# B&R Automation Studio project OpcUaSample410_BrbLibUa103 (part 20)

#### Main.st - Init, cyclic, exit code
```iecst
PROGRAM _INIT
	brsmemset(ADR(Opc), 0, SIZEOF(Opc));
	Opc.OwnGetCertificateList.fbUaSrv_MethodOperate.MethodName := 'OwnGetCertificateList'; // Name der Methode wie in 'Methods.uam' angegeben
	Opc.OwnGenerate.fbUaSrv_MethodOperate.MethodName := 'OwnGenerate'; // Name der Methode wie in 'Methods.uam' angegeben
	Opc.OwnImport.fbUaSrv_MethodOperate.MethodName := 'OwnImport'; // Name der Methode wie in 'Methods.uam' angegeben
	Opc.OwnDelete.fbUaSrv_MethodOperate.MethodName := 'OwnDelete'; // Name der Methode wie in 'Methods.uam' angegeben

	Opc.ForeignGetCertificateList.fbUaSrv_MethodOperate.MethodName := 'ForeignGetCertificateList'; // Name der Methode wie in 'Methods.uam' angegeben
	Opc.ForeignImport.fbUaSrv_MethodOperate.MethodName := 'ForeignImport'; // Name der Methode wie in 'Methods.uam' angegeben
	Opc.ForeignDelete.fbUaSrv_MethodOperate.MethodName := 'ForeignDelete'; // Name der Methode wie in 'Methods.uam' angegeben

	Opc.SslGetCfgList.fbUaSrv_MethodOperate.MethodName := 'SslGetCfgList'; // Name der Methode wie in 'Methods.uam' angegeben
	Opc.SslGetTrustedCertList.fbUaSrv_MethodOperate.MethodName := 'SslGetTrustedCertList'; // Name der Methode wie in 'Methods.uam' angegeben

	Opc.Warmstart.fbUaSrv_MethodOperate.MethodName := 'Warmstart'; // Name der Methode wie in 'Methods.uam' angegeben
END_PROGRAM

PROGRAM _CYCLIC
	// Methode 'OwnGetCertificateList'
	CASE Opc.OwnGetCertificateList.Step.nStepNr OF
		0:	// Prüfen, ob Methode von einem Client aufgerufen wurde
			Opc.OwnGetCertificateList.fbUaSrv_MethodOperate.Execute := 1;
			Opc.OwnGetCertificateList.fbUaSrv_MethodOperate.Action := UaMoa_CheckIsCalled;
			IF Opc.OwnGetCertificateList.fbUaSrv_MethodOperate.Done = 1 THEN
				Opc.OwnGetCertificateList.fbUaSrv_MethodOperate.Execute := 0;
				IF Opc.OwnGetCertificateList.fbUaSrv_MethodOperate.IsCalled = 1 THEN
					// Variablen der Eingans-Argumente sind besetzt -> Methode ausführen
					Opc.OwnGetCertificateList.nCallCount := Opc.OwnGetCertificateList.nCallCount + 1;	// Nur zur Diagnose
					Opc.OwnGetCertificateList.Out_ErrorId := 0;
					Opc.OwnGetCertificateList.Step.nStepNr := Opc.OwnGetCertificateList.Step.nStepNr + 1;
				END_IF
			ELSIF Opc.OwnGetCertificateList.fbUaSrv_MethodOperate.Error = 1 THEN
					Opc.OwnGetCertificateList.fbUaSrv_MethodOperate.Execute := 0;
				Opc.OwnGetCertificateList.Step.nErrorStep := Opc.OwnGetCertificateList.Step.nStepNr;
				Opc.OwnGetCertificateList.Step.eAction := Opc.OwnGetCertificateList.fbUaSrv_MethodOperate.Action;
				Opc.OwnGetCertificateList.Step.nErrorId := Opc.OwnGetCertificateList.fbUaSrv_MethodOperate.ErrorID;
			END_IF

		1:	// Vorbereitung zum Auslesen der Liste
			Opc.OwnGetCertificateList.fbArCertGetOwnDetails.Execute := 0;
			Opc.OwnGetCertificateList.fbArCertGetOwnDetails.Name := '';
			Opc.OwnGetCertificateList.fbArCertGetOwnDetails.Index := 0;
			brsmemset(ADR(Opc.OwnGetCertificateList.Out_CertificatesList), 0, SIZEOF(Opc.OwnGetCertificateList.Out_CertificatesList));
			Opc.OwnGetCertificateList.Step.nStepNr := Opc.OwnGetCertificateList.Step.nStepNr + 1;

		2:	// Nächsten Eintrag auslesen
			IF Opc.OwnGetCertificateList.Out_CertificatesList.nLength <= OPCUA_CERTS_INDEX_MAX THEN
				Opc.OwnGetCertificateList.fbArCertGetOwnDetails.Execute := 1;
				IF Opc.OwnGetCertificateList.fbArCertGetOwnDetails.Busy = 0 THEN
					IF Opc.OwnGetCertificateList.fbArCertGetOwnDetails.Done = 1 THEN
						// Eintrag auf Ausgangs-Argument übertragen
						brsmemcpy(ADR(Opc.OwnGetCertificateList.Out_CertificatesList.Data[Opc.OwnGetCertificateList.Out_CertificatesList.nLength]), ADR(Opc.OwnGetCertificateList.fbArCertGetOwnDetails.Details), SIZEOF(ArCertDetailsType));
						// Nächsten Eintrag lesen
						Opc.OwnGetCertificateList.Out_CertificatesList.nLength := Opc.OwnGetCertificateList.Out_CertificatesList.nLength + 1;
						Opc.OwnGetCertificateList.fbArCertGetOwnDetails.Index := Opc.OwnGetCertificateList.Out_CertificatesList.nLength;
						Opc.OwnGetCertificateList.fbArCertGetOwnDetails.Execute := 0;
					ELSIF Opc.OwnGetCertificateList.fbArCertGetOwnDetails.Error = 1 THEN
						IF Opc.OwnGetCertificateList.fbArCertGetOwnDetails.StatusID = arCERT_ERR_CERTIFICATE_NOT_FOUND THEN
							// Alle Einträge sind gelesen
							Opc.OwnGetCertificateList.fbArCertGetOwnDetails.Execute := 0;
							Opc.OwnGetCertificateList.Step.nStepNr := Opc.OwnGetCertificateList.Step.nStepNr + 1;
						ELSE
							// Fehler beim Auslesen
							Opc.OwnGetCertificateList.fbArCertGetOwnDetails.Execute := 0;
							Opc.OwnGetCertificateList.Out_ErrorId := Opc.OwnGetCertificateList.fbArCertGetOwnDetails.StatusID;
							Opc.OwnGetCertificateList.Step.nStepNr := Opc.OwnGetCertificateList.Step.nStepNr + 1;
						END_IF
					END_IF
				END_IF
			ELSE
				// Das SPS-Array ist nicht genügend groß, um weitere Einträge aufzunehmen
				Opc.OwnGetCertificateList.Out_ErrorId := 12189696; // := 0x00BA0000 := Good_ResultsMayBeIncomplete
				Opc.OwnGetCertificateList.Step.nStepNr := Opc.OwnGetCertificateList.Step.nStepNr + 1;
			END_IF

		3:	// Rückmelden, dass Methode ausgeführt wurde
			Opc.OwnGetCertificateList.fbUaSrv_MethodOperate.Execute := 1;
			Opc.OwnGetCertificateList.fbUaSrv_MethodOperate.Action := UaMoa_Finished;
			IF Opc.OwnGetCertificateList.fbUaSrv_MethodOperate.Done = 1 THEN
				Opc.OwnGetCertificateList.fbUaSrv_MethodOperate.Execute := 0;
				Opc.OwnGetCertificateList.Step.nStepNr := 0;
			ELSIF Opc.OwnGetCertificateList.fbUaSrv_MethodOperate.Error = 1 THEN
				// Fehler eintragen, aber trotzdem weiter machen
				Opc.OwnGetCertificateList.fbUaSrv_MethodOperate.Execute := 0;
				Opc.OwnGetCertificateList.Step.nErrorStep := Opc.OwnGetCertificateList.Step.nStepNr;
				Opc.OwnGetCertificateList.Step.eAction := Opc.OwnGetCertificateList.fbUaSrv_MethodOperate.Action;
				Opc.OwnGetCertificateList.Step.nErrorId := Opc.OwnGetCertificateList.fbUaSrv_MethodOperate.ErrorID;
				Opc.OwnGetCertificateList.Step.nStepNr := 0;
			END_IF

	END_CASE
	Opc.OwnGetCertificateList.fbUaSrv_MethodOperate();
	Opc.OwnGetCertificateList.fbArCertGetOwnDetails();

		// Methode 'OwnGenerate'
	CASE Opc.OwnGenerate.Step.nStepNr OF
		0:	// Prüfen, ob Methode von einem Client aufgerufen wurde
			Opc.OwnGenerate.fbUaSrv_MethodOperate.Execute := 1;
			Opc.OwnGenerate.fbUaSrv_MethodOperate.Action := UaMoa_CheckIsCalled;
			IF Opc.OwnGenerate.fbUaSrv_MethodOperate.Done = 1 THEN
				Opc.OwnGenerate.fbUaSrv_MethodOperate.Execute := 0;
				IF Opc.OwnGenerate.fbUaSrv_MethodOperate.IsCalled = 1 THEN
					// Variablen der Eingans-Argumente sind besetzt -> Methode ausführen
					Opc.OwnGenerate.nCallCount := Opc.OwnGenerate.nCallCount + 1;	// Nur zur Diagnose
					Opc.OwnGenerate.Out_ErrorId := 0;
					Opc.OwnGenerate.Step.nStepNr := Opc.OwnGenerate.Step.nStepNr + 1;
				END_IF
			ELSIF Opc.OwnGenerate.fbUaSrv_MethodOperate.Error = 1 THEN
				Opc.OwnGenerate.fbUaSrv_MethodOperate.Execute := 0;
				Opc.OwnGenerate.Step.nErrorStep := Opc.OwnGenerate.Step.nStepNr;
				Opc.OwnGenerate.Step.eAction := Opc.OwnGenerate.fbUaSrv_MethodOperate.Action;
				Opc.OwnGenerate.Step.nErrorId := Opc.OwnGenerate.fbUaSrv_MethodOperate.ErrorID;
			END_IF

		1:	// Vorbereitung zum Erzeugen des OpcUa-Zertifikats
			Opc.OwnGenerate.fbArCertGenerateX.Execute := 0;
			Opc.OwnGenerate.fbArCertGenerateX.Name := Opc.OwnGenerate.In_Parameter.sName;
			Opc.OwnGenerate.fbArCertGenerateX.PrivateKeyName := Opc.OwnGenerate.In_Parameter.sPrivateKeyName;
			Opc.OwnGenerate.fbArCertGenerateX.PrivateKeyPassword := Opc.OwnGenerate.In_Parameter.sPrivateKeyPassword;
			Opc.OwnGenerate.fbArCertGenerateX.KeySize := Opc.OwnGenerate.In_Parameter.eKeySize;
			Opc.OwnGenerate.fbArCertGenerateX.CountryCode := Opc.OwnGenerate.In_Parameter.sCountryCode;
			Opc.OwnGenerate.fbArCertGenerateX.StateProvince := Opc.OwnGenerate.In_Parameter.sStateProvince;
			Opc.OwnGenerate.fbArCertGenerateX.Locality := Opc.OwnGenerate.In_Parameter.sLocality;
			Opc.OwnGenerate.fbArCertGenerateX.Organization := Opc.OwnGenerate.In_Parameter.sOrganization;
			Opc.OwnGenerate.fbArCertGenerateX.OrganizationUnit := Opc.OwnGenerate.In_Parameter.sOrganizationUnit;
			Opc.OwnGenerate.fbArCertGenerateX.ContactEmail := Opc.OwnGenerate.In_Parameter.sContactEmail;
			Opc.OwnGenerate.fbArCertGenerateX.CommonName := Opc.OwnGenerate.In_Parameter.sCommonName;
			Opc.OwnGenerate.fbArCertGenerateX.ValidTimeSeconds := Opc.OwnGenerate.In_Parameter.nValidTimeSeconds;
			Opc.OwnGenerate.fbArCertGenerateX.URI := Opc.OwnGenerate.In_Parameter.sUri;
			Opc.OwnGenerate.fbArCertGenerateX.DnsName := Opc.OwnGenerate.In_Parameter.sDnsName;
			Opc.OwnGenerate.fbArCertGenerateX.IP := Opc.OwnGenerate.In_Parameter.sIp;
			Opc.OwnGenerate.Step.nStepNr := Opc.OwnGenerate.Step.nStepNr + 1;

		2:	// Erzeugen des OpcUa-Zertifikats
			Opc.OwnGenerate.fbArCertGenerateX.Execute := 1;
			IF Opc.OwnGenerate.fbArCertGenerateX.Busy = 0 THEN
				IF Opc.OwnGenerate.fbArCertGenerateX.Done = 1 THEN
					// Zertifikat wurde erstellt
					Opc.OwnGenerate.fbArCertGenerateX.Execute := 0;
					Opc.OwnGenerate.Step.nStepNr := Opc.OwnGenerate.Step.nStepNr + 1;
				ELSIF Opc.OwnGenerate.fbArCertGenerateX.Error = 1 THEN
					// Fehler beim Erstellen
					Opc.OwnGenerate.fbArCertGenerateX.Execute := 0;
					Opc.OwnGenerate.Out_ErrorId := Opc.OwnGenerate.fbArCertGenerateX.StatusID;
					Opc.OwnGenerate.Step.nStepNr := Opc.OwnGenerate.Step.nStepNr + 1;
				END_IF
			END_IF

		3:	// Rückmelden, dass Methode ausgeführt wurde
			Opc.OwnGenerate.fbUaSrv_MethodOperate.Execute := 1;
			Opc.OwnGenerate.fbUaSrv_MethodOperate.Action := UaMoa_Finished;
			IF Opc.OwnGenerate.fbUaSrv_MethodOperate.Done = 1 THEN
				Opc.OwnGenerate.fbUaSrv_MethodOperate.Execute := 0;
				Opc.OwnGenerate.Step.nStepNr := 0;
			ELSIF Opc.OwnGenerate.fbUaSrv_MethodOperate.Error = 1 THEN
				// Fehler eintragen, aber trotzdem weiter machen
				Opc.OwnGenerate.fbUaSrv_MethodOperate.Execute := 0;
				Opc.OwnGenerate.Step.nErrorStep := Opc.OwnGenerate.Step.nStepNr;
				Opc.OwnGenerate.Step.eAction := Opc.OwnGenerate.fbUaSrv_MethodOperate.Action;
				Opc.OwnGenerate.Step.nErrorId := Opc.OwnGenerate.fbUaSrv_MethodOperate.ErrorID;
				Opc.OwnGenerate.Step.nStepNr := 0;
			END_IF

	END_CASE
	Opc.OwnGenerate.fbUaSrv_MethodOperate();
	Opc.OwnGenerate.fbArCertGenerateX();

	// Methode 'OwnImport'
	CASE Opc.OwnImport.Step.nStepNr OF
		0:	// Prüfen, ob Methode von einem Client aufgerufen wurde
			Opc.OwnImport.fbUaSrv_MethodOperate.Execute := 1;
			Opc.OwnImport.fbUaSrv_MethodOperate.Action := UaMoa_CheckIsCalled;
			IF Opc.OwnImport.fbUaSrv_MethodOperate.Done = 1 THEN
				Opc.OwnImport.fbUaSrv_MethodOperate.Execute := 0;
				IF Opc.OwnImport.fbUaSrv_MethodOperate.IsCalled = 1 THEN
					// Variablen der Eingans-Argumente sind besetzt -> Methode ausführen
					Opc.OwnImport.nCallCount := Opc.OwnImport.nCallCount + 1;	// Nur zur Diagnose
					Opc.OwnImport.Out_ErrorId := 0;
					Opc.OwnImport.Step.nStepNr := Opc.OwnImport.Step.nStepNr + 1;
				END_IF
			ELSIF Opc.OwnImport.fbUaSrv_MethodOperate.Error = 1 THEN
				Opc.OwnImport.fbUaSrv_MethodOperate.Execute := 0;
				Opc.OwnImport.Step.nErrorStep := Opc.OwnImport.Step.nStepNr;
				Opc.OwnImport.Step.eAction := Opc.OwnImport.fbUaSrv_MethodOperate.Action;
				Opc.OwnImport.Step.nErrorId := Opc.OwnImport.fbUaSrv_MethodOperate.ErrorID;
			END_IF

		1:	// Vorbereitung zum Löschen des öffentlichen Zertifikats
			Opc.OwnImport.fbArCertDeleteOwn.Execute := 0;
			IF Opc.OwnImport.In_Overwrite = 1 THEN
				Opc.OwnImport.fbArCertDeleteOwn.Name := Opc.OwnImport.In_Name;
				Opc.OwnImport.Step.nStepNr := Opc.OwnImport.Step.nStepNr + 1;
			ELSE
				Opc.OwnImport.Step.nStepNr := Opc.OwnImport.Step.nStepNr + 2;
			END_IF

		2:	// Löschen des öffentlichen Zertifikats
			Opc.OwnImport.fbArCertDeleteOwn.Execute := 1;
			IF Opc.OwnImport.fbArCertDeleteOwn.Busy = 0 THEN
				IF Opc.OwnImport.fbArCertDeleteOwn.Done = 1 THEN
					// Zertifikat wurde gelöscht
					Opc.OwnImport.fbArCertDeleteOwn.Execute := 0;
					Opc.OwnImport.Step.nStepNr := Opc.OwnImport.Step.nStepNr + 1;
				ELSIF Opc.OwnImport.fbArCertDeleteOwn.Error = 1 THEN
					// Zertifikat ist nicht vorhanden. Fehler wird übergangen
					Opc.OwnImport.fbArCertDeleteOwn.Execute := 0;
					Opc.OwnImport.Step.nStepNr := Opc.OwnImport.Step.nStepNr + 1;
				END_IF
			END_IF

		3:	// Vorbereitung zum Importieren des öffentlichen Zertifikats
			Opc.OwnImport.fbArCertImportOwn.Execute := 0;
			Opc.OwnImport.fbArCertImportOwn.Name := Opc.OwnImport.In_Name;
			Opc.OwnImport.fbArCertImportOwn.Data := ADR(Opc.OwnImport.In_Certificate.Data);
			Opc.OwnImport.fbArCertImportOwn.DataSize := Opc.OwnImport.In_Certificate.Length;
			Opc.OwnImport.Step.nStepNr := Opc.OwnImport.Step.nStepNr + 1;

		4:	// Importieren des öffentlichen Zertifikats
			Opc.OwnImport.fbArCertImportOwn.Execute := 1;
			IF Opc.OwnImport.fbArCertImportOwn.Busy = 0 THEN
				IF Opc.OwnImport.fbArCertImportOwn.Done = 1 THEN
					// Zertifikat wurde importiert
					Opc.OwnImport.fbArCertImportOwn.Execute := 0;
					Opc.OwnImport.Step.nStepNr := Opc.OwnImport.Step.nStepNr + 1;
				ELSIF Opc.OwnImport.fbArCertImportOwn.Error = 1 THEN
					// Fehler beim Importieren
					Opc.OwnImport.fbArCertImportOwn.Execute := 0;
					Opc.OwnImport.Out_ErrorId := Opc.OwnImport.fbArCertImportOwn.StatusID;
					Opc.OwnImport.Step.nStepNr := Opc.OwnImport.Step.nStepNr + 1;
				END_IF
			END_IF

		5:	// Vorbereitung zum Löschen des privaten Keys
			Opc.OwnImport.fbArCertDeletePrivateKey.Execute := 0;
			IF Opc.OwnImport.In_Overwrite = 1 THEN
				Opc.OwnImport.fbArCertDeletePrivateKey.Name := Opc.OwnImport.In_PrivateKeyName;
				Opc.OwnImport.Step.nStepNr := Opc.OwnImport.Step.nStepNr + 1;
			ELSE
				Opc.OwnImport.Step.nStepNr := Opc.OwnImport.Step.nStepNr + 2;
			END_IF

		6:	// Löschen des privaten Keys
			Opc.OwnImport.fbArCertDeletePrivateKey.Execute := 1;
			IF Opc.OwnImport.fbArCertDeletePrivateKey.Busy = 0 THEN
				IF Opc.OwnImport.fbArCertDeletePrivateKey.Done = 1 THEN
					// Key wurde gelöscht
					Opc.OwnImport.fbArCertDeletePrivateKey.Execute := 0;
					Opc.OwnImport.Step.nStepNr := Opc.OwnImport.Step.nStepNr + 1;
				ELSIF Opc.OwnImport.fbArCertDeletePrivateKey.Error = 1 THEN
				// Key ist nicht vorhanden. Fehler wird übergangen
					Opc.OwnImport.fbArCertDeleteOwn.Execute := 0;
					Opc.OwnImport.Step.nStepNr := Opc.OwnImport.Step.nStepNr + 1;
				END_IF
			END_IF

		7:	// Vorbereitung zum Importieren des privaten Keys
			Opc.OwnImport.fbArCertImportPrivateKey.Execute := 0;
			Opc.OwnImport.fbArCertImportPrivateKey.Name := Opc.OwnImport.In_PrivateKeyName;
			Opc.OwnImport.fbArCertImportPrivateKey.Data := ADR(Opc.OwnImport.In_PrivateKey.Data);
			Opc.OwnImport.fbArCertImportPrivateKey.DataSize := Opc.OwnImport.In_PrivateKey.Length;
			Opc.OwnImport.Step.nStepNr := Opc.OwnImport.Step.nStepNr + 1;

		8:	// Importieren des privaten Keys
			Opc.OwnImport.fbArCertImportPrivateKey.Execute := 1;
			IF Opc.OwnImport.fbArCertImportPrivateKey.Busy = 0 THEN
				IF Opc.OwnImport.fbArCertImportPrivateKey.Done = 1 THEN
				// Key wurde importiert
					Opc.OwnImport.fbArCertImportPrivateKey.Execute := 0;
					Opc.OwnImport.Step.nStepNr := Opc.OwnImport.Step.nStepNr + 1;
				ELSIF Opc.OwnImport.fbArCertImportPrivateKey.Error = 1 THEN
				// Fehler beim Importieren
					Opc.OwnImport.fbArCertImportPrivateKey.Execute := 0;
					Opc.OwnImport.Out_ErrorId := Opc.OwnImport.fbArCertImportPrivateKey.StatusID;
					Opc.OwnImport.Step.nStepNr := Opc.OwnImport.Step.nStepNr + 1;
				END_IF
			END_IF

		9:	// Rückmelden, dass Methode ausgeführt wurde
			Opc.OwnImport.fbUaSrv_MethodOperate.Execute := 1;
			Opc.OwnImport.fbUaSrv_MethodOperate.Action := UaMoa_Finished;
			IF Opc.OwnImport.fbUaSrv_MethodOperate.Done = 1 THEN
				Opc.OwnImport.fbUaSrv_MethodOperate.Execute := 0;
				Opc.OwnImport.Step.nStepNr := 0;
			ELSIF Opc.OwnImport.fbUaSrv_MethodOperate.Error = 1 THEN
				// Fehler eintragen, aber trotzdem weiter machen
				Opc.OwnImport.fbUaSrv_MethodOperate.Execute := 0;
				Opc.OwnImport.Step.nErrorStep := Opc.OwnImport.Step.nStepNr;
				Opc.OwnImport.Step.eAction := Opc.OwnImport.fbUaSrv_MethodOperate.Action;
				Opc.OwnImport.Step.nErrorId := Opc.OwnImport.fbUaSrv_MethodOperate.ErrorID;
				Opc.OwnImport.Step.nStepNr := 0;
			END_IF

	END_CASE
	Opc.OwnImport.fbUaSrv_MethodOperate();
	Opc.OwnImport.fbArCertDeleteOwn();
	Opc.OwnImport.fbArCertImportOwn();
	Opc.OwnImport.fbArCertDeletePrivateKey();
	Opc.OwnImport.fbArCertImportPrivateKey();

	// Methode 'OwnDelete'
	CASE Opc.OwnDelete.Step.nStepNr OF
		0:	// Prüfen, ob Methode von einem Client aufgerufen wurde
			Opc.OwnDelete.fbUaSrv_MethodOperate.Execute := 1;
			Opc.OwnDelete.fbUaSrv_MethodOperate.Action := UaMoa_CheckIsCalled;
			IF Opc.OwnDelete.fbUaSrv_MethodOperate.Done = 1 THEN
				Opc.OwnDelete.fbUaSrv_MethodOperate.Execute := 0;
				IF Opc.OwnDelete.fbUaSrv_MethodOperate.IsCalled = 1 THEN
					// Variablen der Eingans-Argumente sind besetzt -> Methode ausführen
					Opc.OwnDelete.nCallCount := Opc.OwnDelete.nCallCount + 1;	// Nur zur Diagnose
					Opc.OwnDelete.Out_ErrorId := 0;
					Opc.OwnDelete.Step.nStepNr := Opc.OwnDelete.Step.nStepNr + 1;
				END_IF
			ELSIF Opc.OwnDelete.fbUaSrv_MethodOperate.Error = 1 THEN
				Opc.OwnDelete.fbUaSrv_MethodOperate.Execute := 0;
				Opc.OwnDelete.Step.nErrorStep := Opc.OwnDelete.Step.nStepNr;
				Opc.OwnDelete.Step.eAction := Opc.OwnDelete.fbUaSrv_MethodOperate.Action;
				Opc.OwnDelete.Step.nErrorId := Opc.OwnDelete.fbUaSrv_MethodOperate.ErrorID;
			END_IF

		1:	// Vorbereitung zum Löschen des öffentlichen Zertifikats
			Opc.OwnDelete.fbArCertDeleteOwn.Execute := 0;
			IF brsstrlen(ADR(Opc.OwnDelete.In_Name)) > 0 THEN
				Opc.OwnDelete.fbArCertDeleteOwn.Name := Opc.OwnDelete.In_Name;
				Opc.OwnDelete.Step.nStepNr := Opc.OwnDelete.Step.nStepNr + 1;
			ELSE
				Opc.OwnDelete.Step.nStepNr := Opc.OwnDelete.Step.nStepNr + 2;
			END_IF

		2:	// Löschen des öffentlichen Zertifikats
			Opc.OwnDelete.fbArCertDeleteOwn.Execute := 1;
			IF Opc.OwnDelete.fbArCertDeleteOwn.Busy = 0 THEN
				IF Opc.OwnDelete.fbArCertDeleteOwn.Done = 1 THEN
					// Zertifikat wurde gelöscht
					Opc.OwnDelete.fbArCertDeleteOwn.Execute := 0;
					Opc.OwnDelete.Step.nStepNr := Opc.OwnDelete.Step.nStepNr + 1;
				ELSIF Opc.OwnDelete.fbArCertDeleteOwn.Error = 1 THEN
					IF Opc.OwnDelete.fbArCertDeleteOwn.StatusID = arCERT_ERR_CERTIFICATE_NOT_FOUND AND Opc.OwnDelete.In_SuppressNotExistsError = 1 THEN
						// Fehler 'Certificate not found' soll unterdrückt werden
						Opc.OwnDelete.fbArCertDeleteOwn.Execute := 0;
						Opc.OwnDelete.Step.nStepNr := Opc.OwnDelete.Step.nStepNr + 1;
					ELSE
						// Fehler beim Löschen
						Opc.OwnDelete.fbArCertDeleteOwn.Execute := 0;
						Opc.OwnDelete.Out_ErrorId := Opc.OwnDelete.fbArCertDeleteOwn.StatusID;
						Opc.OwnDelete.Step.nStepNr := Opc.OwnDelete.Step.nStepNr + 1;
					END_IF
				END_IF
			END_IF

		3:	// Vorbereitung zum Löschen des privaten Keys
			Opc.OwnDelete.fbArCertDeletePrivateKey.Execute := 0;
			IF brsstrlen(ADR(Opc.OwnDelete.In_PrivateKeyName)) > 0 THEN
				Opc.OwnDelete.fbArCertDeletePrivateKey.Name := Opc.OwnDelete.In_PrivateKeyName;
				Opc.OwnDelete.Step.nStepNr := Opc.OwnDelete.Step.nStepNr + 1;
			ELSE
				Opc.OwnDelete.Step.nStepNr := Opc.OwnDelete.Step.nStepNr + 2;
			END_IF

		4:	// Löschen des privaten Keys
			Opc.OwnDelete.fbArCertDeletePrivateKey.Execute := 1;
			IF Opc.OwnDelete.fbArCertDeletePrivateKey.Busy = 0 THEN
				IF Opc.OwnDelete.fbArCertDeletePrivateKey.Done = 1 THEN
					// Zertifikat wurde gelöscht
					Opc.OwnDelete.fbArCertDeletePrivateKey.Execute := 0;
					Opc.OwnDelete.Step.nStepNr := Opc.OwnDelete.Step.nStepNr + 1;
				ELSIF Opc.OwnDelete.fbArCertDeletePrivateKey.Error = 1 THEN
					IF Opc.OwnDelete.fbArCertDeletePrivateKey.StatusID = arCERT_ERR_CERTIFICATE_NOT_FOUND AND Opc.OwnDelete.In_SuppressNotExistsError = 1 THEN
						// Fehler 'Certificate not found' soll unterdrückt werden
						Opc.OwnDelete.fbArCertDeletePrivateKey.Execute := 0;
						Opc.OwnDelete.Step.nStepNr := Opc.OwnDelete.Step.nStepNr + 1;
					ELSE
						// Fehler beim Löschen
						Opc.OwnDelete.fbArCertDeletePrivateKey.Execute := 0;
						Opc.OwnDelete.Out_ErrorId := Opc.OwnDelete.fbArCertDeletePrivateKey.StatusID;
						Opc.OwnDelete.Step.nStepNr := Opc.OwnDelete.Step.nStepNr + 1;
					END_IF
				END_IF
			END_IF

		5:	// Rückmelden, dass Methode ausgeführt wurde
			Opc.OwnDelete.fbUaSrv_MethodOperate.Execute := 1;
			Opc.OwnDelete.fbUaSrv_MethodOperate.Action := UaMoa_Finished;
			IF Opc.OwnDelete.fbUaSrv_MethodOperate.Done = 1 THEN
				Opc.OwnDelete.fbUaSrv_MethodOperate.Execute := 0;
				Opc.OwnDelete.Step.nStepNr := 0;
			ELSIF Opc.OwnDelete.fbUaSrv_MethodOperate.Error = 1 THEN
				// Fehler eintragen, aber trotzdem weiter machen
				Opc.OwnDelete.fbUaSrv_MethodOperate.Execute := 0;
				Opc.OwnDelete.Step.nErrorStep := Opc.OwnDelete.Step.nStepNr;
				Opc.OwnDelete.Step.eAction := Opc.OwnDelete.fbUaSrv_MethodOperate.Action;
				Opc.OwnDelete.Step.nErrorId := Opc.OwnDelete.fbUaSrv_MethodOperate.ErrorID;
				Opc.OwnDelete.Step.nStepNr := 0;
			END_IF

	END_CASE
	Opc.OwnDelete.fbUaSrv_MethodOperate();
	Opc.OwnDelete.fbArCertDeleteOwn();
	Opc.OwnDelete.fbArCertDeletePrivateKey();

	// Methode 'ForeignGetCertificateList'
	CASE Opc.ForeignGetCertificateList.Step.nStepNr OF
		0:	// Prüfen, ob Methode von einem Client aufgerufen wurde
			Opc.ForeignGetCertificateList.fbUaSrv_MethodOperate.Execute := 1;
			Opc.ForeignGetCertificateList.fbUaSrv_MethodOperate.Action := UaMoa_CheckIsCalled;
			IF Opc.ForeignGetCertificateList.fbUaSrv_MethodOperate.Done = 1 THEN
				Opc.ForeignGetCertificateList.fbUaSrv_MethodOperate.Execute := 0;
				IF Opc.ForeignGetCertificateList.fbUaSrv_MethodOperate.IsCalled = 1 THEN
					// Variablen der Eingans-Argumente sind besetzt -> Methode ausführen
					Opc.ForeignGetCertificateList.nCallCount := Opc.ForeignGetCertificateList.nCallCount + 1;	// Nur zur Diagnose
					Opc.ForeignGetCertificateList.Out_ErrorId := 0;
					Opc.ForeignGetCertificateList.Step.nStepNr := Opc.ForeignGetCertificateList.Step.nStepNr + 1;
				END_IF
			ELSIF Opc.ForeignGetCertificateList.fbUaSrv_MethodOperate.Error = 1 THEN
				Opc.ForeignGetCertificateList.fbUaSrv_MethodOperate.Execute := 0;
				Opc.ForeignGetCertificateList.Step.nErrorStep := Opc.ForeignGetCertificateList.Step.nStepNr;
				Opc.ForeignGetCertificateList.Step.eAction := Opc.ForeignGetCertificateList.fbUaSrv_MethodOperate.Action;
				Opc.ForeignGetCertificateList.Step.nErrorId := Opc.ForeignGetCertificateList.fbUaSrv_MethodOperate.ErrorID;
			END_IF

		1:	// Vorbereitung zum Auslesen der Liste
			Opc.ForeignGetCertificateList.fbArCertGetThirdPartyDetails.Execute := 0;
			Opc.ForeignGetCertificateList.fbArCertGetThirdPartyDetails.Name := '';
			Opc.ForeignGetCertificateList.fbArCertGetThirdPartyDetails.Index := 0;
			brsmemset(ADR(Opc.ForeignGetCertificateList.Out_CertificatesList), 0, SIZEOF(Opc.ForeignGetCertificateList.Out_CertificatesList));
			Opc.ForeignGetCertificateList.Step.nStepNr := Opc.ForeignGetCertificateList.Step.nStepNr + 1;

		2:	// Nächsten Eintrag auslesen
			IF Opc.ForeignGetCertificateList.Out_CertificatesList.nLength <= OPCUA_CERTS_INDEX_MAX THEN
				Opc.ForeignGetCertificateList.fbArCertGetThirdPartyDetails.Execute := 1;
				IF Opc.ForeignGetCertificateList.fbArCertGetThirdPartyDetails.Busy = 0 THEN
					IF Opc.ForeignGetCertificateList.fbArCertGetThirdPartyDetails.Done = 1 THEN
						// Eintrag auf Ausgangs-Argument übertragen
						brsmemcpy(ADR(Opc.ForeignGetCertificateList.Out_CertificatesList.Data[Opc.ForeignGetCertificateList.Out_CertificatesList.nLength]), ADR(Opc.ForeignGetCertificateList.fbArCertGetThirdPartyDetails.Details), SIZEOF(ArCertDetailsType));
						// Nächsten Eintrag lesen
						Opc.ForeignGetCertificateList.Out_CertificatesList.nLength := Opc.ForeignGetCertificateList.Out_CertificatesList.nLength + 1;
						Opc.ForeignGetCertificateList.fbArCertGetThirdPartyDetails.Index := Opc.ForeignGetCertificateList.Out_CertificatesList.nLength;
						Opc.ForeignGetCertificateList.fbArCertGetThirdPartyDetails.Execute := 0;
					ELSIF Opc.ForeignGetCertificateList.fbArCertGetThirdPartyDetails.Error = 1 THEN
						IF Opc.ForeignGetCertificateList.fbArCertGetThirdPartyDetails.StatusID = arCERT_ERR_CERTIFICATE_NOT_FOUND THEN
							// Alle Einträge sind gelesen
							Opc.ForeignGetCertificateList.fbArCertGetThirdPartyDetails.Execute := 0;
							Opc.ForeignGetCertificateList.Step.nStepNr := Opc.ForeignGetCertificateList.Step.nStepNr + 1;
						ELSE
							// Fehler beim Auslesen
							Opc.ForeignGetCertificateList.fbArCertGetThirdPartyDetails.Execute := 0;
							Opc.ForeignGetCertificateList.Out_ErrorId := Opc.ForeignGetCertificateList.fbArCertGetThirdPartyDetails.StatusID;
							Opc.ForeignGetCertificateList.Step.nStepNr := Opc.ForeignGetCertificateList.Step.nStepNr + 1;
						END_IF
					END_IF
				END_IF
			ELSE
				// Das SPS-Array ist nicht genügend groß, um weitere Einträge aufzunehmen
				Opc.ForeignGetCertificateList.Out_ErrorId := 12189696; // := 0x00BA0000 := Good_ResultsMayBeIncomplete
				Opc.ForeignGetCertificateList.Step.nStepNr := Opc.ForeignGetCertificateList.Step.nStepNr + 1;
			END_IF

		3:	// Rückmelden, dass Methode ausgeführt wurde
			Opc.ForeignGetCertificateList.fbUaSrv_MethodOperate.Execute := 1;
			Opc.ForeignGetCertificateList.fbUaSrv_MethodOperate.Action := UaMoa_Finished;
			IF Opc.ForeignGetCertificateList.fbUaSrv_MethodOperate.Done = 1 THEN
				Opc.ForeignGetCertificateList.fbUaSrv_MethodOperate.Execute := 0;
				Opc.ForeignGetCertificateList.Step.nStepNr := 0;
			ELSIF Opc.ForeignGetCertificateList.fbUaSrv_MethodOperate.Error = 1 THEN
				// Fehler eintragen, aber trotzdem weiter machen
				Opc.ForeignGetCertificateList.fbUaSrv_MethodOperate.Execute := 0;
				Opc.ForeignGetCertificateList.Step.nErrorStep := Opc.ForeignGetCertificateList.Step.nStepNr;
				Opc.ForeignGetCertificateList.Step.eAction := Opc.ForeignGetCertificateList.fbUaSrv_MethodOperate.Action;
				Opc.ForeignGetCertificateList.Step.nErrorId := Opc.ForeignGetCertificateList.fbUaSrv_MethodOperate.ErrorID;
				Opc.ForeignGetCertificateList.Step.nStepNr := 0;
			END_IF

	END_CASE
	Opc.ForeignGetCertificateList.fbUaSrv_MethodOperate();
	Opc.ForeignGetCertificateList.fbArCertGetThirdPartyDetails();

	// Methode 'ForeignImport'
	CASE Opc.ForeignImport.Step.nStepNr OF
		0:	// Prüfen, ob Methode von einem Client aufgerufen wurde
			Opc.ForeignImport.fbUaSrv_MethodOperate.Execute := 1;
			Opc.ForeignImport.fbUaSrv_MethodOperate.Action := UaMoa_CheckIsCalled;
			IF Opc.ForeignImport.fbUaSrv_MethodOperate.Done = 1 THEN
				Opc.ForeignImport.fbUaSrv_MethodOperate.Execute := 0;
				IF Opc.ForeignImport.fbUaSrv_MethodOperate.IsCalled = 1 THEN
					// Variablen der Eingans-Argumente sind besetzt -> Methode ausführen
					Opc.ForeignImport.nCallCount := Opc.ForeignImport.nCallCount + 1;	// Nur zur Diagnose
					Opc.ForeignImport.Out_ErrorId := 0;
					Opc.ForeignImport.Step.nStepNr := Opc.ForeignImport.Step.nStepNr + 1;
				END_IF
			ELSIF Opc.ForeignImport.fbUaSrv_MethodOperate.Error = 1 THEN
				Opc.ForeignImport.fbUaSrv_MethodOperate.Execute := 0;
				Opc.ForeignImport.Step.nErrorStep := Opc.ForeignImport.Step.nStepNr;
				Opc.ForeignImport.Step.eAction := Opc.ForeignImport.fbUaSrv_MethodOperate.Action;
				Opc.ForeignImport.Step.nErrorId := Opc.ForeignImport.fbUaSrv_MethodOperate.ErrorID;
			END_IF

		1:	// Vorbereitung zum Löschen des öffentlichen Zertifikats
			Opc.ForeignImport.fbArCertDeleteThirdParty.Execute := 0;
			IF Opc.ForeignImport.In_Overwrite = 1 THEN
				Opc.ForeignImport.fbArCertDeleteThirdParty.Name := Opc.ForeignImport.In_Name;
				Opc.ForeignImport.Step.nStepNr := Opc.ForeignImport.Step.nStepNr + 1;
			ELSE
				Opc.ForeignImport.Step.nStepNr := Opc.ForeignImport.Step.nStepNr + 2;
			END_IF

		2:	// Löschen des öffentlichen Zertifikats
			Opc.ForeignImport.fbArCertDeleteThirdParty.Execute := 1;
			IF Opc.ForeignImport.fbArCertDeleteThirdParty.Busy = 0 THEN
				IF Opc.ForeignImport.fbArCertDeleteThirdParty.Done = 1 THEN
					// Zertifikat wurde gelöscht
					Opc.ForeignImport.fbArCertDeleteThirdParty.Execute := 0;
					Opc.ForeignImport.Step.nStepNr := Opc.ForeignImport.Step.nStepNr + 1;
				ELSIF Opc.ForeignImport.fbArCertDeleteThirdParty.Error = 1 THEN
					// Zertifikat ist nicht vorhanden. Fehler wird übergangen
					Opc.ForeignImport.fbArCertDeleteThirdParty.Execute := 0;
					Opc.ForeignImport.Step.nStepNr := Opc.ForeignImport.Step.nStepNr + 1;
				END_IF
			END_IF

		3:	// Vorbereitung zum Importieren des öffentlichen Zertifikats
			Opc.ForeignImport.fbArCertImportThirdParty.Execute := 0;
			Opc.ForeignImport.fbArCertImportThirdParty.Name := Opc.ForeignImport.In_Name;
			Opc.ForeignImport.fbArCertImportThirdParty.Data := ADR(Opc.ForeignImport.In_Certificate.Data);
			Opc.ForeignImport.fbArCertImportThirdParty.DataSize := Opc.ForeignImport.In_Certificate.Length;
			Opc.ForeignImport.Step.nStepNr := Opc.ForeignImport.Step.nStepNr + 1;

		4:	// Importieren des öffentlichen Zertifikats
			Opc.ForeignImport.fbArCertImportThirdParty.Execute := 1;
			IF Opc.ForeignImport.fbArCertImportThirdParty.Busy = 0 THEN
				IF Opc.ForeignImport.fbArCertImportThirdParty.Done = 1 THEN
					// Zertifikat wurde importiert
					Opc.ForeignImport.fbArCertImportThirdParty.Execute := 0;
					Opc.ForeignImport.Step.nStepNr := Opc.ForeignImport.Step.nStepNr + 1;
				ELSIF Opc.ForeignImport.fbArCertImportThirdParty.Error = 1 THEN
					// Fehler beim Importieren
					Opc.ForeignImport.fbArCertImportThirdParty.Execute := 0;
					Opc.ForeignImport.Out_ErrorId := Opc.ForeignImport.fbArCertImportThirdParty.StatusID;
					Opc.ForeignImport.Step.nStepNr := Opc.ForeignImport.Step.nStepNr + 1;
				END_IF
			END_IF

		5:	// Rückmelden, dass Methode ausgeführt wurde
			Opc.ForeignImport.fbUaSrv_MethodOperate.Execute := 1;
			Opc.ForeignImport.fbUaSrv_MethodOperate.Action := UaMoa_Finished;
			IF Opc.ForeignImport.fbUaSrv_MethodOperate.Done = 1 THEN
				Opc.ForeignImport.fbUaSrv_MethodOperate.Execute := 0;
				Opc.ForeignImport.Step.nStepNr := 0;
			ELSIF Opc.ForeignImport.fbUaSrv_MethodOperate.Error = 1 THEN
				// Fehler eintragen, aber trotzdem weiter machen
				Opc.ForeignImport.fbUaSrv_MethodOperate.Execute := 0;
				Opc.ForeignImport.Step.nErrorStep := Opc.ForeignImport.Step.nStepNr;
				Opc.ForeignImport.Step.eAction := Opc.ForeignImport.fbUaSrv_MethodOperate.Action;
				Opc.ForeignImport.Step.nErrorId := Opc.ForeignImport.fbUaSrv_MethodOperate.ErrorID;
				Opc.ForeignImport.Step.nStepNr := 0;
			END_IF

	END_CASE
	Opc.ForeignImport.fbUaSrv_MethodOperate();
	Opc.ForeignImport.fbArCertDeleteThirdParty();
	Opc.ForeignImport.fbArCertImportThirdParty();

	// Methode 'ForeignDelete'
	CASE Opc.ForeignDelete.Step.nStepNr OF
		0:	// Prüfen, ob Methode von einem Client aufgerufen wurde
			Opc.ForeignDelete.fbUaSrv_MethodOperate.Execute := 1;
			Opc.ForeignDelete.fbUaSrv_MethodOperate.Action := UaMoa_CheckIsCalled;
			IF Opc.ForeignDelete.fbUaSrv_MethodOperate.Done = 1 THEN
				Opc.ForeignDelete.fbUaSrv_MethodOperate.Execute := 0;
				IF Opc.ForeignDelete.fbUaSrv_MethodOperate.IsCalled = 1 THEN
					// Variablen der Eingans-Argumente sind besetzt -> Methode ausführen
					Opc.ForeignDelete.nCallCount := Opc.ForeignDelete.nCallCount + 1;	// Nur zur Diagnose
					Opc.ForeignDelete.Out_ErrorId := 0;
					Opc.ForeignDelete.Step.nStepNr := Opc.ForeignDelete.Step.nStepNr + 1;
				END_IF
			ELSIF Opc.ForeignDelete.fbUaSrv_MethodOperate.Error = 1 THEN
				Opc.ForeignDelete.fbUaSrv_MethodOperate.Execute := 0;
				Opc.ForeignDelete.Step.nErrorStep := Opc.ForeignDelete.Step.nStepNr;
				Opc.ForeignDelete.Step.eAction := Opc.ForeignDelete.fbUaSrv_MethodOperate.Action;
				Opc.ForeignDelete.Step.nErrorId := Opc.ForeignDelete.fbUaSrv_MethodOperate.ErrorID;
			END_IF

		1:	// Vorbereitung zum Löschen des öffentlichen Zertifikats
			Opc.ForeignDelete.fbArCertDeleteThirdParty.Execute := 0;
			IF brsstrlen(ADR(Opc.ForeignDelete.In_Name)) > 0 THEN
				Opc.ForeignDelete.fbArCertDeleteThirdParty.Name := Opc.ForeignDelete.In_Name;
				Opc.ForeignDelete.Step.nStepNr := Opc.ForeignDelete.Step.nStepNr + 1;
			ELSE
				Opc.ForeignDelete.Step.nStepNr := Opc.ForeignDelete.Step.nStepNr + 2;
			END_IF

		2:	// Löschen des öffentlichen Zertifikats
			Opc.ForeignDelete.fbArCertDeleteThirdParty.Execute := 1;
			IF Opc.ForeignDelete.fbArCertDeleteThirdParty.Busy = 0 THEN
				IF Opc.ForeignDelete.fbArCertDeleteThirdParty.Done = 1 THEN
					// Zertifikat wurde gelöscht
					Opc.ForeignDelete.fbArCertDeleteThirdParty.Execute := 0;
					Opc.ForeignDelete.Step.nStepNr := Opc.ForeignDelete.Step.nStepNr + 1;
				ELSIF Opc.ForeignDelete.fbArCertDeleteThirdParty.Error = 1 THEN
					IF Opc.ForeignDelete.fbArCertDeleteThirdParty.StatusID = arCERT_ERR_CERTIFICATE_NOT_FOUND AND Opc.ForeignDelete.In_SuppressNotExistsError = 1 THEN
						// Fehler 'Certificate not found' soll unterdrückt werden
						Opc.ForeignDelete.fbArCertDeleteThirdParty.Execute := 0;
						Opc.ForeignDelete.Step.nStepNr := Opc.ForeignDelete.Step.nStepNr + 1;
					ELSE
					// Fehler beim Löschen
						Opc.ForeignDelete.fbArCertDeleteThirdParty.Execute := 0;
						Opc.ForeignDelete.Out_ErrorId := Opc.ForeignDelete.fbArCertDeleteThirdParty.StatusID;
						Opc.ForeignDelete.Step.nStepNr := Opc.ForeignDelete.Step.nStepNr + 1;
					END_IF
				END_IF
			END_IF

		3:	// Rückmelden, dass Methode ausgeführt wurde
			Opc.ForeignDelete.fbUaSrv_MethodOperate.Execute := 1;
			Opc.ForeignDelete.fbUaSrv_MethodOperate.Action := UaMoa_Finished;
			IF Opc.ForeignDelete.fbUaSrv_MethodOperate.Done = 1 THEN
				Opc.ForeignDelete.fbUaSrv_MethodOperate.Execute := 0;
				Opc.ForeignDelete.Step.nStepNr := 0;
			ELSIF Opc.ForeignDelete.fbUaSrv_MethodOperate.Error = 1 THEN
				// Fehler eintragen, aber trotzdem weiter machen
				Opc.ForeignDelete.fbUaSrv_MethodOperate.Execute := 0;
				Opc.ForeignDelete.Step.nErrorStep := Opc.ForeignDelete.Step.nStepNr;
				Opc.ForeignDelete.Step.eAction := Opc.ForeignDelete.fbUaSrv_MethodOperate.Action;
				Opc.ForeignDelete.Step.nErrorId := Opc.ForeignDelete.fbUaSrv_MethodOperate.ErrorID;
				Opc.ForeignDelete.Step.nStepNr := 0;
			END_IF

	END_CASE
	Opc.ForeignDelete.fbUaSrv_MethodOperate();
	Opc.ForeignDelete.fbArCertDeleteThirdParty();

	// Methode 'SslGetCfgList'
	CASE Opc.SslGetCfgList.Step.nStepNr OF
		0:	// Prüfen, ob Methode von einem Client aufgerufen wurde
			Opc.SslGetCfgList.fbUaSrv_MethodOperate.Execute := 1;
			Opc.SslGetCfgList.fbUaSrv_MethodOperate.Action := UaMoa_CheckIsCalled;
			IF Opc.SslGetCfgList.fbUaSrv_MethodOperate.Done = 1 THEN
				Opc.SslGetCfgList.fbUaSrv_MethodOperate.Execute := 0;
				IF Opc.SslGetCfgList.fbUaSrv_MethodOperate.IsCalled = 1 THEN
					// Variablen der Eingans-Argumente sind besetzt -> Methode ausführen
					Opc.SslGetCfgList.nCallCount := Opc.SslGetCfgList.nCallCount + 1;	// Nur zur Diagnose
					Opc.SslGetCfgList.Out_ErrorId := 0;
					Opc.SslGetCfgList.Step.nStepNr := Opc.SslGetCfgList.Step.nStepNr + 1;
				END_IF
			ELSIF Opc.SslGetCfgList.fbUaSrv_MethodOperate.Error = 1 THEN
				Opc.SslGetCfgList.fbUaSrv_MethodOperate.Execute := 0;
				Opc.SslGetCfgList.Step.nErrorStep := Opc.SslGetCfgList.Step.nStepNr;
				Opc.SslGetCfgList.Step.eAction := Opc.SslGetCfgList.fbUaSrv_MethodOperate.Action;
				Opc.SslGetCfgList.Step.nErrorId := Opc.SslGetCfgList.fbUaSrv_MethodOperate.ErrorID;
			END_IF

		1:	// Vorbereitung zum Auslesen der Cfg-Liste
			Opc.SslGetCfgList.fbArSslGetCfgDetails.Execute := 0;
			Opc.SslGetCfgList.fbArSslGetCfgDetails.Name := '';
			Opc.SslGetCfgList.fbArSslGetCfgDetails.Index := 0;
			brsmemset(ADR(Opc.SslGetCfgList.Out_CfgList), 0, SIZEOF(Opc.SslGetCfgList.Out_CfgList));
			Opc.SslGetCfgList.Step.nStepNr := Opc.SslGetCfgList.Step.nStepNr + 1;

		2:	// Nächsten Cfg-Eintrag auslesen
			IF Opc.SslGetCfgList.Out_CfgList.nLength <= OPCUA_SSLCFG_INDEX_MAX THEN
				Opc.SslGetCfgList.fbArSslGetCfgDetails.Execute := 1;
				IF Opc.SslGetCfgList.fbArSslGetCfgDetails.Busy = 0 THEN
					IF Opc.SslGetCfgList.fbArSslGetCfgDetails.Done = 1 THEN
						// Cfg-Eintrag auf Ausgangs-Argument übertragen
						brsmemcpy(ADR(Opc.SslGetCfgList.Out_CfgList.Data[Opc.SslGetCfgList.Out_CfgList.nLength]), ADR(Opc.SslGetCfgList.fbArSslGetCfgDetails.Details), SIZEOF(ArSslCfgDetailsType));
						// Nächsten Eintrag lesen
						Opc.SslGetCfgList.Out_CfgList.nLength := Opc.SslGetCfgList.Out_CfgList.nLength + 1;
						Opc.SslGetCfgList.fbArSslGetCfgDetails.Index := Opc.SslGetCfgList.Out_CfgList.nLength;
						Opc.SslGetCfgList.fbArSslGetCfgDetails.Execute := 0;
					ELSIF Opc.SslGetCfgList.fbArSslGetCfgDetails.Error = 1 THEN
						IF Opc.SslGetCfgList.fbArSslGetCfgDetails.StatusID = arSSL_ERR_SSL_CFG_NOT_FOUND THEN
							// Alle Cfg-Einträge sind gelesen
							Opc.SslGetCfgList.fbArSslGetCfgDetails.Execute := 0;
							Opc.SslGetCfgList.Step.nStepNr := Opc.SslGetCfgList.Step.nStepNr + 1;
						ELSE
							// Fehler beim Auslesen
							Opc.SslGetCfgList.fbArSslGetCfgDetails.Execute := 0;
							Opc.SslGetCfgList.Out_ErrorId := Opc.SslGetCfgList.fbArSslGetCfgDetails.StatusID;
							Opc.SslGetCfgList.Step.nStepNr := Opc.SslGetCfgList.Step.nStepNr + 1;
						END_IF
					END_IF
				END_IF
			ELSE
				// Das SPS-Array ist nicht genügend groß, um weitere Einträge aufzunehmen
				Opc.SslGetCfgList.Out_ErrorId := 12189696; // := 0x00BA0000 := Good_ResultsMayBeIncomplete
				Opc.SslGetCfgList.Step.nStepNr := Opc.SslGetCfgList.Step.nStepNr + 1;
			END_IF

		3:	// Rückmelden, dass Methode ausgeführt wurde
			Opc.SslGetCfgList.fbUaSrv_MethodOperate.Execute := 1;
			Opc.SslGetCfgList.fbUaSrv_MethodOperate.Action := UaMoa_Finished;
			IF Opc.SslGetCfgList.fbUaSrv_MethodOperate.Done = 1 THEN
				Opc.SslGetCfgList.fbUaSrv_MethodOperate.Execute := 0;
				Opc.SslGetCfgList.Step.nStepNr := 0;
			ELSIF Opc.SslGetCfgList.fbUaSrv_MethodOperate.Error = 1 THEN
				// Fehler eintragen, aber trotzdem weiter machen
				Opc.SslGetCfgList.fbUaSrv_MethodOperate.Execute := 0;
				Opc.SslGetCfgList.Step.nErrorStep := Opc.SslGetCfgList.Step.nStepNr;
				Opc.SslGetCfgList.Step.eAction := Opc.SslGetCfgList.fbUaSrv_MethodOperate.Action;
				Opc.SslGetCfgList.Step.nErrorId := Opc.SslGetCfgList.fbUaSrv_MethodOperate.ErrorID;
				Opc.SslGetCfgList.Step.nStepNr := 0;
			END_IF

	END_CASE
	Opc.SslGetCfgList.fbUaSrv_MethodOperate();
	Opc.SslGetCfgList.fbArSslGetCfgDetails();

	// Methode 'SslGetTrustedCertList'
	CASE Opc.SslGetTrustedCertList.Step.nStepNr OF
		0:	// Prüfen, ob Methode von einem Client aufgerufen wurde
			Opc.SslGetTrustedCertList.fbUaSrv_MethodOperate.Execute := 1;
			Opc.SslGetTrustedCertList.fbUaSrv_MethodOperate.Action := UaMoa_CheckIsCalled;
			IF Opc.SslGetTrustedCertList.fbUaSrv_MethodOperate.Done = 1 THEN
				Opc.SslGetTrustedCertList.fbUaSrv_MethodOperate.Execute := 0;
				IF Opc.SslGetTrustedCertList.fbUaSrv_MethodOperate.IsCalled = 1 THEN
					// Variablen der Eingans-Argumente sind besetzt -> Methode ausführen
					Opc.SslGetTrustedCertList.nCallCount := Opc.SslGetTrustedCertList.nCallCount + 1;	// Nur zur Diagnose
					Opc.SslGetTrustedCertList.Out_ErrorId := 0;
					Opc.SslGetTrustedCertList.Step.nStepNr := Opc.SslGetTrustedCertList.Step.nStepNr + 1;
				END_IF
			ELSIF Opc.SslGetTrustedCertList.fbUaSrv_MethodOperate.Error = 1 THEN
				Opc.SslGetTrustedCertList.fbUaSrv_MethodOperate.Execute := 0;
				Opc.SslGetTrustedCertList.Step.nErrorStep := Opc.SslGetTrustedCertList.Step.nStepNr;
				Opc.SslGetTrustedCertList.Step.eAction := Opc.SslGetTrustedCertList.fbUaSrv_MethodOperate.Action;
				Opc.SslGetTrustedCertList.Step.nErrorId := Opc.SslGetTrustedCertList.fbUaSrv_MethodOperate.ErrorID;
			END_IF

		1:	// Vorbereitung zum Auslesen der Liste
			Opc.SslGetTrustedCertList.fbArSslGetCertificate.Execute := 0;
			Opc.SslGetTrustedCertList.fbArSslGetCertificate.Name := Opc.SslGetTrustedCertList.In_CfgName;
			Opc.SslGetTrustedCertList.fbArSslGetCertificate.Index := 0;
			brsmemset(ADR(Opc.SslGetTrustedCertList.Out_TrustedCertNameList), 0, SIZEOF(Opc.SslGetTrustedCertList.Out_TrustedCertNameList));
			Opc.SslGetTrustedCertList.Step.nStepNr := Opc.SslGetTrustedCertList.Step.nStepNr + 1;

		2:	// Nächsten Eintrag auslesen
			IF Opc.SslGetTrustedCertList.Out_TrustedCertNameList.nLength <= OPCUA_CERTS_INDEX_MAX THEN
				Opc.SslGetTrustedCertList.fbArSslGetCertificate.Execute := 1;
				IF Opc.SslGetTrustedCertList.fbArSslGetCertificate.Busy = 0 THEN
					IF Opc.SslGetTrustedCertList.fbArSslGetCertificate.Done = 1 THEN
						// Eintrag auf Ausgangs-Argument übertragen
						Opc.SslGetTrustedCertList.Out_TrustedCertNameList.Data[Opc.SslGetTrustedCertList.Out_TrustedCertNameList.nLength] := Opc.SslGetTrustedCertList.fbArSslGetCertificate.TrustedCertificate;
						// Nächsten Eintrag lesen
						Opc.SslGetTrustedCertList.Out_TrustedCertNameList.nLength := Opc.SslGetTrustedCertList.Out_TrustedCertNameList.nLength + 1;
						Opc.SslGetTrustedCertList.fbArSslGetCertificate.Index := Opc.SslGetTrustedCertList.Out_TrustedCertNameList.nLength;
						Opc.SslGetTrustedCertList.fbArSslGetCertificate.Execute := 0;
					ELSIF Opc.SslGetTrustedCertList.fbArSslGetCertificate.Error = 1 THEN
						IF Opc.SslGetTrustedCertList.fbArSslGetCertificate.StatusID = arSSL_ERR_INDEX_OUT_OF_RANGE THEN
							// Alle Einträge sind gelesen
							Opc.SslGetTrustedCertList.fbArSslGetCertificate.Execute := 0;
							Opc.SslGetTrustedCertList.Step.nStepNr := Opc.SslGetTrustedCertList.Step.nStepNr + 1;
						ELSE
							// Fehler beim Auslesen
							Opc.SslGetTrustedCertList.fbArSslGetCertificate.Execute := 0;
							Opc.SslGetTrustedCertList.Out_ErrorId := Opc.SslGetTrustedCertList.fbArSslGetCertificate.StatusID;
							Opc.SslGetTrustedCertList.Step.nStepNr := Opc.SslGetTrustedCertList.Step.nStepNr + 1;
						END_IF
					END_IF
				END_IF
			ELSE
				// Das SPS-Array ist nicht genügend groß, um weitere Einträge aufzunehmen
				Opc.SslGetTrustedCertList.Out_ErrorId := 12189696; // := 0x00BA0000 := Good_ResultsMayBeIncomplete
				Opc.SslGetTrustedCertList.Step.nStepNr := Opc.SslGetTrustedCertList.Step.nStepNr + 1;
			END_IF

		3:	// Rückmelden, dass Methode ausgeführt wurde
			Opc.SslGetTrustedCertList.fbUaSrv_MethodOperate.Execute := 1;
			Opc.SslGetTrustedCertList.fbUaSrv_MethodOperate.Action := UaMoa_Finished;
			IF Opc.SslGetTrustedCertList.fbUaSrv_MethodOperate.Done = 1 THEN
				Opc.SslGetTrustedCertList.fbUaSrv_MethodOperate.Execute := 0;
				Opc.SslGetTrustedCertList.Step.nStepNr := 0;
			ELSIF Opc.SslGetTrustedCertList.fbUaSrv_MethodOperate.Error = 1 THEN
				// Fehler eintragen, aber trotzdem weiter machen
				Opc.SslGetTrustedCertList.fbUaSrv_MethodOperate.Execute := 0;
				Opc.SslGetTrustedCertList.Step.nErrorStep := Opc.SslGetTrustedCertList.Step.nStepNr;
				Opc.SslGetTrustedCertList.Step.eAction := Opc.SslGetTrustedCertList.fbUaSrv_MethodOperate.Action;
				Opc.SslGetTrustedCertList.Step.nErrorId := Opc.SslGetTrustedCertList.fbUaSrv_MethodOperate.ErrorID;
				Opc.SslGetTrustedCertList.Step.nStepNr := 0;
			END_IF

	END_CASE
	Opc.SslGetTrustedCertList.fbUaSrv_MethodOperate();
	Opc.SslGetTrustedCertList.fbArSslGetCertificate();

	// Methode 'Warmstart'
	CASE Opc.Warmstart.Step.nStepNr OF
		0:	// Prüfen, ob Methode von einem Client aufgerufen wurde
			Opc.Warmstart.fbUaSrv_MethodOperate.Execute := 1;
			Opc.Warmstart.fbUaSrv_MethodOperate.Action := UaMoa_CheckIsCalled;
			IF Opc.Warmstart.fbUaSrv_MethodOperate.Done = 1 THEN
				Opc.Warmstart.fbUaSrv_MethodOperate.Execute := 0;
				IF Opc.Warmstart.fbUaSrv_MethodOperate.IsCalled = 1 THEN
					// Variablen der Eingans-Argumente sind besetzt -> Methode ausführen
					Opc.Warmstart.nCallCount := Opc.Warmstart.nCallCount + 1;	// Nur zur Diagnose
					Opc.Warmstart.Step.nStepNr := Opc.Warmstart.Step.nStepNr + 1;
				END_IF
			ELSIF Opc.Warmstart.fbUaSrv_MethodOperate.Error = 1 THEN
				Opc.Warmstart.fbUaSrv_MethodOperate.Execute := 0;
				Opc.Warmstart.Step.nErrorStep := Opc.Warmstart.Step.nStepNr;
				Opc.Warmstart.Step.eAction := Opc.Warmstart.fbUaSrv_MethodOperate.Action;
				Opc.Warmstart.Step.nErrorId := Opc.Warmstart.fbUaSrv_MethodOperate.ErrorID;
			END_IF

		1:	// Verzögerung für das Auslösen des Warmstarts starten
			// Der Warmstart wird verzögert ausgelöst, damit vom Server die Rückmeldung noch geschickt werden kann
			Opc.Warmstart.fbTon.PT := t#2s;
			Opc.Warmstart.fbTon.IN := 1;
			Opc.Warmstart.Step.nStepNr := Opc.Warmstart.Step.nStepNr + 1;

		2:	// Rückmelden, dass Methode ausgeführt wurde
			Opc.Warmstart.fbUaSrv_MethodOperate.Execute := 1;
			Opc.Warmstart.fbUaSrv_MethodOperate.Action := UaMoa_Finished;
			IF Opc.Warmstart.fbUaSrv_MethodOperate.Done = 1 THEN
				Opc.Warmstart.fbUaSrv_MethodOperate.Execute := 0;
				Opc.Warmstart.Step.nStepNr := 0;
			ELSIF Opc.Warmstart.fbUaSrv_MethodOperate.Error = 1 THEN
				// Fehler eintragen, aber trotzdem weiter machen
				Opc.Warmstart.fbUaSrv_MethodOperate.Execute := 0;
				Opc.Warmstart.Step.nErrorStep := Opc.Warmstart.Step.nStepNr;
				Opc.Warmstart.Step.eAction := Opc.Warmstart.fbUaSrv_MethodOperate.Action;
				Opc.Warmstart.Step.nErrorId := Opc.Warmstart.fbUaSrv_MethodOperate.ErrorID;
				Opc.Warmstart.Step.nStepNr := 0;
			END_IF

	END_CASE
	Opc.Warmstart.fbUaSrv_MethodOperate();
	Opc.Warmstart.fbTon();
	IF Opc.Warmstart.fbTon.Q = 1 THEN
		Opc.Warmstart.fbTon.IN := 0;
		SYSreset(1, 1); // Warmstart auslösen
	END_IF
END_PROGRAM

PROGRAM _EXIT
END_PROGRAM
```

#### Types.typ - Local data types
```iecst
TYPE
	Step_TYP : 	STRUCT
		nStepNr : DINT;
		nErrorStep : DINT;
		eAction : UaMethodOperateAction;
		nErrorId : DWORD;
	END_STRUCT;
	OpcUaCertList_TYP : 	STRUCT
		nLength : UAArrayLength;
		Data : ARRAY[0..9]OF ArCertDetailsType; (*OPCUA_CERTS_INDEX_MAX*)
	END_STRUCT;
	OwnGetCertificateList_TYP : 	STRUCT
		Step : Step_TYP;
		fbUaSrv_MethodOperate : UaSrv_MethodOperate;
		nCallCount : UDINT;
		fbArCertGetOwnDetails : ArCertGetOwnDetails;
		Out_CertificatesList : OpcUaCertList_TYP;
		Out_ErrorId : DINT;
	END_STRUCT;
	OwnGenerateCertificatePar_TYP : 	STRUCT
		sName : STRING[255];
		sPrivateKeyName : STRING[255];
		sPrivateKeyPassword : STRING[255];
		eKeySize : ArCertKeySizeEnum;
		sCountryCode : STRING[9];
		sStateProvince : STRING[513];
		sLocality : STRING[513];
		sOrganization : STRING[255];
		sOrganizationUnit : STRING[255];
		sContactEmail : STRING[513];
		sCommonName : STRING[255];
		nValidTimeSeconds : UDINT;
		sUri : STRING[513];
		sDnsName : STRING[513];
		sIp : STRING[513];
	END_STRUCT;
	OwnGenerateCertificate_TYP : 	STRUCT
		Step : Step_TYP;
		fbUaSrv_MethodOperate : UaSrv_MethodOperate;
		nCallCount : UDINT;
		fbArCertGenerateX : ArCertGenerateX;
		In_Parameter : OwnGenerateCertificatePar_TYP;
		Out_ErrorId : DINT;
	END_STRUCT;
	UAByteString5k_TYP : 	STRUCT
		Length : DINT;
		Data : ARRAY[0..4999]OF USINT;
	END_STRUCT;
	OwnImportCertificate_TYP : 	STRUCT
		Step : Step_TYP;
		fbUaSrv_MethodOperate : UaSrv_MethodOperate;
		nCallCount : UDINT;
		fbArCertDeleteOwn : ArCertDeleteOwn;
		fbArCertImportOwn : ArCertImportOwn;
		fbArCertDeletePrivateKey : ArCertDeletePrivateKey;
		fbArCertImportPrivateKey : ArCertImportPrivateKey;
		In_Name : STRING[255];
		In_Certificate : UAByteString5k_TYP;
		In_PrivateKeyName : STRING[255];
		In_PrivateKey : UAByteString5k_TYP;
		In_Overwrite : BOOL;
		Out_ErrorId : DINT;
	END_STRUCT;
	OwnDeleteCertificate_TYP : 	STRUCT
		Step : Step_TYP;
		fbUaSrv_MethodOperate : UaSrv_MethodOperate;
		nCallCount : UDINT;
		fbArCertDeleteOwn : ArCertDeleteOwn;
		fbArCertDeletePrivateKey : ArCertDeletePrivateKey;
		In_Name : STRING[255];
		In_PrivateKeyName : STRING[255];
		In_SuppressNotExistsError : BOOL;
		Out_ErrorId : DINT;
	END_STRUCT;
	ForeignGetCertificateList_TYP : 	STRUCT
		Step : Step_TYP;
		fbUaSrv_MethodOperate : UaSrv_MethodOperate;
		nCallCount : UDINT;
		fbArCertGetThirdPartyDetails : ArCertGetThirdPartyDetails;
		Out_CertificatesList : OpcUaCertList_TYP;
		Out_ErrorId : DINT;
	END_STRUCT;
	ForeignImportCertificate_TYP : 	STRUCT
		Step : Step_TYP;
		fbUaSrv_MethodOperate : UaSrv_MethodOperate;
		nCallCount : UDINT;
		fbArCertDeleteThirdParty : ArCertDeleteThirdParty;
		fbArCertImportThirdParty : ArCertImportThirdParty;
		In_Name : STRING[255];
		In_Certificate : UAByteString5k_TYP;
		In_Overwrite : BOOL;
		Out_ErrorId : DINT;
	END_STRUCT;
	ForeignDeleteCertificate_TYP : 	STRUCT
		Step : Step_TYP;
		fbUaSrv_MethodOperate : UaSrv_MethodOperate;
		nCallCount : UDINT;
		fbArCertDeleteThirdParty : ArCertDeleteThirdParty;
		In_Name : STRING[255];
		In_SuppressNotExistsError : BOOL;
		Out_ErrorId : DINT;
	END_STRUCT;
	OpcUaSslCfgList_TYP : 	STRUCT
		nLength : UAArrayLength;
		Data : ARRAY[0..9]OF ArSslCfgDetailsType; (*OPCUA_SSLCFG_INDEX_MAX*)
	END_STRUCT;
	SslGetCfgList_TYP : 	STRUCT
		Step : Step_TYP;
		fbUaSrv_MethodOperate : UaSrv_MethodOperate;
		nCallCount : UDINT;
		fbArSslGetCfgDetails : ArSslGetCfgDetails;
		Out_CfgList : OpcUaSslCfgList_TYP;
		Out_ErrorId : DINT;
	END_STRUCT;
	OpcUaCertNameList_TYP : 	STRUCT
		nLength : UAArrayLength;
		Data : ARRAY[0..9]OF STRING[255]; (*OPCUA_CERTS_INDEX_MAX*)
	END_STRUCT;
	SslGetTrustedCertList_TYP : 	STRUCT
		Step : Step_TYP;
		fbUaSrv_MethodOperate : UaSrv_MethodOperate;
		nCallCount : UDINT;
		fbArSslGetCertificate : ArSslGetCertificate;
		In_CfgName : STRING[255];
		Out_TrustedCertNameList : OpcUaCertNameList_TYP;
		Out_ErrorId : DINT;
	END_STRUCT;
	Warmstart_TYP : 	STRUCT
		Step : Step_TYP;
		fbUaSrv_MethodOperate : UaSrv_MethodOperate;
		nCallCount : UDINT;
		fbTon : TON;
	END_STRUCT;
	Opc_TYP : 	STRUCT
		OwnGetCertificateList : OwnGetCertificateList_TYP;
		OwnGenerate : OwnGenerateCertificate_TYP;
		OwnImport : OwnImportCertificate_TYP;
		OwnDelete : OwnDeleteCertificate_TYP;
		ForeignGetCertificateList : ForeignGetCertificateList_TYP;
		ForeignImport : ForeignImportCertificate_TYP;
		ForeignDelete : ForeignDeleteCertificate_TYP;
		SslGetCfgList : SslGetCfgList_TYP;
		SslGetTrustedCertList : SslGetTrustedCertList_TYP;
		Warmstart : Warmstart_TYP;
	END_STRUCT;
END_TYPE
```

#### Variables.var - Local variables
```iecst
VAR CONSTANT
	OPCUA_CERTS_INDEX_MAX : UINT := 9;
	OPCUA_SSLCFG_INDEX_MAX : UINT := 9;
END_VAR
VAR
	Opc : Opc_TYP;
END_VAR
```

### Package Logical/Tasks/AirCond - Klima-Anlagen: Eigenes Daten-Modell

### ReadMe.txt
```
Mit diesem Beispiel wird verdeutlicht, wie eigene oder extern definierte OpcUa-Modelle eingesetzt werden können.
	Hinweis: Um die implementierten Modelle zu betrachten und besser zu verstehen, sollte mit einem Test-Client
	(z.B. UaExpert oder RnCommTest) eine Verbindung aufgebaut und der Adress-Raum gebrowst werden.

Erklärung der Task-Funktionalität:
	Als funktionelles Beispiel dient die Implementierung mehrerer Instanzen einer Klima-Anlage.
	Es gibt einen Typ Klima-Anlage, dessen Daten in der Struktur "AirCond_TYP" aufgelegt sind:
		AirCond_TYP
			sName																	Name der Instanz
			Act																		Ist-Werte
				eOperationMode											Betriebs-Modus (0=Aus, 1=Manuell, 2=Automatik)
				rTemperature												Ist-Temperatur in [°C]
				nFanLevel														Ist-Lüfter-Stufe (0-5, 0=Aus)
			Set																		Soll-Werte
				rTemperature												Soll-Temperatur in [°C] für Automatik
				nFanLevel														Soll-Lüfter-Stufe (0-5, 0=Aus) für Manuell

	Es gibt drei Instanzen: Schlafzimmer, Flur und Wohnzimmer. Für jede dieser Instanzen werden die
	entsprechenden Funktionen "Init", "Operate" und "Simulation" aufgerufen. Das bedeutet, dass der
	Code einer Klima-Anlage nur einmal vorhanden ist und Änderung daran nur an einer Stelle gemacht
	werden müssen.
	Jede dieser Instanzen ist im OpcUa-Model mit entsprechenden Rechten freigegeben (siehe Configuration View
	unter "../PC/Connectivity/OpcUA/OpcUaMap.uad").
	Zusätzlich gibt es für jede Klima-Anlagen-Instanz auch noch eine Struktur-Variable "AirCondIntern_TYP". Sie
	enthält Elemente, die als Variablen für die interne Behandlung einer Instanz nötig sind (z.B.
	Schrittketten-Zähler), welche aber nicht über OpcUa freigegeben sind.

	Hier nun die Beschreibung der einzelnen Funktionen, welche für jede Instanz aufgerufen werden:
	Init: Die Werte einer Instanz werden hier vorbesetzt.

	Steuerung:
		Betriebsmodus:
			Aus:
				Der Lüfter bleibt ausgeschaltet (Stufe=0).
			Manuell:
				Der Lüfter wird auf die im Sollwert angegebene Stufe gesetzt.
			Automatik:
				Die Lüfter-Stufe wird aufgrund der prozentualen Abweichung zwischen Ist- und Soll-Wert gesetzt.
		Ausserdem wird hier in einer Schrittkette der Methoden-Aufruf für "SetOperationMode" behandelt.
		Es gibt auch eine Schrittkette, die das Feuern eines Events beim Ändern des Betriebsmodus behandelt.

	Simulation:
		Die Ist-Temperatur wird ständig erhöht und drängt dadurch auf 26.0°C.
		Je nach Lüfter-Stufe wird die Ist-Temperatur abgesenkt und wirkt dadurch der natürlichen
		Erwärmung entgegen.
		Die Ist-Temperatur wird auf den Bereich 15.0 - 26.0°C begrenzt, um ein Abdriften zu verhindern.

	OpcUa-Methode "SetOperationMode":
		Die Methode setzt den Betriebsmodus, welcher als einziges Eingangs-Argument übergeben wird.
		Als Ausgangs-Argument wird ein applikativer Status zurückgegeben, welcher auf einen ungültigen
		Betriebsmodus hinweisen kann (dies ist eigentlich nicht möglich, da der Betriebsmodus als Enumeration
		aufgelegt ist).

	OpcUa-Event "AirConditionOperationModeChanged":
		Bei jeder Änderung des Betriebsmodus wird ein Event gefeuert, welches als zusätzliche Felder die
		Informationen 'OldOperationMode' und 'NewOperationMode' besitzt.

OpcUa-Methode(n) "SetOperationMode":
	In "Methods.uam" ist für jede Instanz jeweils die Methode "SetOperationMode" deklariert. So wird garantiert,
	dass bei jeder Instanz diese Methode gleichzeitig zu den anderen Instanzen aufgerufen werden kann.
	Die Schrittkette für diese Methode ist nur einmal implementiert und wird für jede Instanz einzeln aufgerufen
	(siehe oben).

OpcUa-Event(s) "AirConditionOperationModeChanged":
	Dieses Event wurde eigens für dieses Beispiel modelliert und ist im Fremd-Modell hinterlegt (siehe
	'/Root/Types/EventTypes/BaseEventType/AirConditionOperationModeChanged').
	Normalerweise (wie auch hier) können alle am Server gefeuerten Events durch Abonnierung des Knotens
	'/Root/Objects/Server' (i=2253)	von einem Client empfangen werden. In dieses Beispiel wurde eine zusätzliche
	Möglichkeit implementiert:
	Auch der Instanz-Knoten einer Klima-Anlage im Fremd-Modell (z.B. 'BedRoom') soll abonniert werden können,
	aber nur das Event der betreffenden Instanz feuern.
	Der meiste Teil dieser Anforderung muss im Modeller umgesetzt werden. Im Sps-Programm ist nur eines wichtig:
	Beim Feuern des Events muss das Feld 'SourceNode' applikativ mit der NodeId des Hauptknotens besetzt werden
	(also z.B. 'ns=6;i=5013' für 'BedRoom' in der ANSI-C-Variante).
	Hinweis: Ob ein Knoten Events feuern und deswegen abonniert werden kann, lässt sich sehr leicht mit dem
	Attribut 'EventNotifier' des Knotens prüfen. Es ist bitcodiert. Ist Bit#0 (=SubscribeToEvents) gesetzt,
	so kann der Knoten auf Events abonniert werden.

OpcUa-Modelle:
	Im B&R-Modell, das automatisch vom Compiler erzeugt und vom OpcUa-Server veröffentlicht wird, werden die
	drei Instanzen und deren Methoden in der Ebene des Tasks angezeigt:
		Root
		+--	Objects
				+--	PLC (hier beginnt das automatisch erzeugte B&R-Modell)
						+--	Modules
								+--	Default
										+--	AirCondC (dies ist der Task)
												+--	BedRoomSetOperationMode (Methode)
												+--	CorridorSetOperationMode (Methode)
												+--	LivingRoomSetOperationMode (Methode)
												+--	AirCond_BedRoom (Daten)
												|		+-- Act (Ist-Werte)
												|		|		+--	eOperationMode
												|		|		+--	nFanLevel
												|		|		+--	rTemperature
												|		+--	Set (Soll-Werte)
												|		|		+--	nFanLevel
												|		|		+--	rTemperature
												|		+--	sName (Name der Instanz)
												+--	AirCond_Corridor (Daten)
												|		+-- ...
												+--	AirCond_LivingRoom (Daten)
														+-- ...

	Es kann nun aber eine andere Hierarchie der Knoten gewünscht sein. In diesem Beispiel soll die Vorgabe
	sein, dass es jeweils einen Knoten pro Instanz gibt, der die Daten und die dazugehörige Methode enthält.
	Dieser Knoten soll auch das Event feuern können. Auch die Namen der Knoten sollen anders sein (keine
	Präfixe).
	Dazu wurde ein eigenes Modell definiert, das diese Vorgaben erfüllt. Da	dieses Beispiel Tasks sowohl für
	ANSI-C als auch für StructureText enthält, wurde auch im Modell diese	Aufteilung berücksichtigt. Hier das
	Modell für ANSI-C:

		Root
		+--	Objects
				+--	DeviceSet
						+--	AirConditions (hier beginnt das eigene Modell)
								+--	C	(ANSI-C-Variante)
										+--	BedRoom
										|		+--	SetOperationMode (Methode)
										|		+-- Act (Ist-Werte)
										|		|		+--	FanLevel
										|		|		+--	OperationMode
										|		|		+--	Temperature
										|		+--	Name (Name der Instanz)
										|		+--	Set (Soll-Werte)
										|				+--	FanLevel
										|				+--	Temperature
										+--	Corridor
										|		+-- ...
										+--	LivingRoom
												+-- ...

	Dieser Zweig des Modells musste in einem externen Modeler-Tool definiert werden. Momentan gibt es keine
	Möglichkeit, dies im AS zu tun. Hier wurde das Tool "UaModeler" der Fa. Unified Automation verwendet.
	Hinweis: Die übliche Praxis sieht vor, Datentypen und Instanzen der Knoten jeweils in separaten Modellen
	zu halten. Der Einfachkeit halber wurde in diesem Beispiel alles in ein Modell gepackt.
	Diese neuen Knoten können über das von der Foundation standardisierte Opc-Export-Format "nodeset" ins AS
	importiert werden. Dies geschieht im AS in der Configuration View unter dem Zweig
	"../PC/Connectivity/OpcUA/". Für dieses Beispiel ist es die Datei "aircondmodel.uanodeset", welche aus
	dem externen Model-Tool exportiert wurde.
	Diese neuen Knoten haben von sich aus aber keine Werte, sie hängen praktisch "in der Luft". Deshalb gibt es
	die Möglichkeit, solche Knoten an bereits bestehende B&R-Knoten zu "mappen" und diese so mit derselben
	Funktionalität zu versehen wie der gemappte Knoten.
	Dieses Mapping geschieht durch OpcUa-Referenzen. B&R hat hierzu eigene Referenz-Typen implementiert.
	Variablen:
		Durch die Referenz "BrHasValueAttribute" kann ein Knoten auf einen bestehenden Variablen-Knoten aus dem
		B&R-Modell gemappt werden.
	Methoden:
		Analog dazu gibt es die Referenz "BrHasImplementation", mit der auf einen bestehenden Methoden-Knoten aus dem
		B&R-Modell gemappt werden kann.
	Dies bedeutet für den B&R-Server, diesen neuen Knoten genauso zu behandeln wie den gemappten Knoten.

	Mapping:
		Bis AS4.6 musste das Setzen der Vorwärts-Referenzen ebenfalls im externen Modeler-Tool gemacht werden.
		Ab AS4.7 ist es möglich, eine Rückwärts-Referenz aus dem B&R-Modell ins neu importierte eigene Modell zu setzen.
		Dies hat den Vorteil, dass das externe Modell für das Mapping nicht mehr geändert werden muss.
		Beim Kompilieren des Projekts werden dann automatisch die Vorwärts-Referenzen für die Knoten im externen
		Modell gebildet.
		Das Setzen der Rückwärts-Referenzen geschieht in der Datei 'OpcUaMap.uad', in dem auch alle sonstigen Knoten-
		Einstellungen gemacht werden.

		Zuerst müssen die im externen Modell verwendeten Namespaces angegeben werden. Dies geschieht in den
		Eigenschaften	des obersten Knotens 'Default View'. Hier gibt es eine Liste 'Namespaces URIs', welche von Haus
		aus die vom	B&R-Modell verwendeten Namespaces enthält. Die Liste muss nun mit den im eigenen Modell verwendeten
		Namespaces erweitert werden. In unserem Fall ist dies nur einer mit dem Namen
		'http://br-automation.com/AirCondModel/' (so wurde es im externen Model definiert) mit dem Namespace-Index 5.

		Zum Mappen der Knoten gibt es jetzt einen Parameter 'Reference/Value Attribute Of' für Variablen-Knoten und
		'Reference/Implementation Of' für Methoden-Knoten in den Eigenschaften des Knotens. Hier muss textuell die
		NodeId auf den zu mappenden Knoten des eigenen Modells gesetzt werden (z.B.
		'ns=5;i=6041'). Dadurch wird der Knoten des externen Modells genauso behandelt wie der Knoten im B&R-Modell.
		Als Namespace-Index muss der aus der obigen Liste verwendet werden. Achtung: Der Namespace-Index wird vom
		Server zur Laufzeit automatisch neu vergeben.

	Namespace-Indizes bei Verwendung eigener/externer Modelle:
		Namespace-Uri's von externen Modellen müssen angegeben werden. Bei der Parametrierung von Referenzen im AS muss
		der Namespace-Index dieser Liste angegeben werden (siehe oben).
		Die in dieser Liste angegebenen Indizes sind NICHT die zur Laufzeit verwendeten Namespace-Indizes!
		Zur Laufzeit werden die Namespaces erneut zusammengeführt und erhalten so andere Namespace-Indizes!
		In unserem Beispiel liegt der neue Namespace 'http://br-automation.com/AirCondModel/' auf dem Namespace-
		Index 6. Der Namespace-Index des B&R-Modells verschiebt sich daher auf 7! Dies muss bei allen Verwendungen
		von NodeId's/Browsepfaden auf das B&R-Modell berücksichtigt werden, auch bei allen externen Clients!
		In diesem Beispiel-Projekt war es daher nötig, die Browse-Pfade bei der Konfiguration des OpcUaAny-Clients
		anzupassen.
		Diese Verschiebung des B&R-Namespace-Index durch externe Modelle wird in einer der nächsten	AS-Versionen behoben
		sein, so dass der B&R-Index auf 6 bleiben wird.

	Erleichterung gegenüber AS4.6
		Damit im externen Modell die Vorwärts-Referenzen gesetzt werden konnten (bis AS4.6), musste das vom AS
		erzeugte B&R-Modell in das Modeler-Tool importiert werden. Dies war zwar sehr einfach, jedoch konnte ein einmal
		importiertes B&R-Modell nicht ohne weiters nochmals importiert werden, wenn sich dieses geändert hatte.
		Durch das Setzen der Referenzen im AS4.7 braucht das B&R-Modell gar nicht mehr im UaModeler importiert zu
		werden.

	Verwendung von Datentypen/Enumerationen im externen Modell:
		Dass das B&R-Modell im Modeler-Tool nicht bekannt ist, hat aber auch einen Nachteil: Im B&R-Projekt definierte
		Datentypen und Enumerationen sind dann im externen Modell nicht bekannt und können damit auch nicht in den
		neuen Knoten verwendet werden.
		In unserem Beispiel betrifft das die zwei Enumerationen:

			AirCondOperationMode_ENUM
				Dies ist die Aufzählung der Betriebsmodi für eine Klima-Anlage:
					eAC_OPERATIONMODE_OFF						0
					eAC_OPERATIONMODE_MANUAL				1
					eAC_OPERATIONMODE_AUTO					2
				Sie wird beim Modell benötigt für:
					-Variable 'Act.OperationMode'
					-Eingangs-Argument bei Methode 'SetOperationMode'
					-Felder des Events 'AirConditionOperationModeChanged'
				Natürlich könnten diese Knoten im externen Modell als Int32 deklariert werden, was aber den Vorteil einer
				Enumeration unter OpcUa zunichte macht:
					-Anzeige von Texten anstatt Zahlen
					-Definierte Grenzen (0..2) bei der Eingabe
				Um die Vorteile einer Enumeration trotzdem zu nutzen, ohne das B&R-Modell zu importieren, wurde folgende
				Alternative gewählt: Im externen Modell wurde ein eigener Enumerations-Datentyp angelegt, der der
				Definition im B&R-Projekt entspricht. Unter dem Pfad 'Root/Types/DataTypes/BaseDataType/Enumeration/' gibt
				es nun den Enumerations-Knoten 'AirConditionOperationModeType', der folgende Elemente enthält:
					Off															0
					Manual													1
					Automatic												2
				Dieser wird nun als Datentyp für die Variablen/Argumente/Felder verwendet.

			AirCondMethodStatus_ENUM
				Dies ist die Aufzählung für den Status einer 'SetOperationMode'-Methode:
					eAC_METH_STATUS_OK							0
					eAC_METH_STATUS_INVALID_OPMODE	1
				Sie wird beim Modell benötigt für das Ausgangs-Argument bei Methode 'SetOperationMode'.
				Auch hier wurde dieselbe Alternative gewählt: Im externen Modell wurde ein eigener Enumerations-Datentyp
				angelegt, der der	Definition im B&R-Projekt entspricht. Unter dem Pfad
				'Root/Types/DataTypes/BaseDataType/Enumeration/' gibt	es nun den Enumerations-Knoten
				'AirConditionMethodStatusType', der folgende Elemente enthält:
					Ok															0
					InvalidOperationMode						1
				Dieser wird nun als Datentyp für das Argument verwendet.

			Übrigens ist dies eine übliche Praxis: Die im Fremd-Modell angelegten Datentypen und Enumerationen sind
			auf der Sps 'nachgebaut' und umgekehrt.

	Ordner 'UaModeler'
		In diesem Ordner des Packages sind die Dateien enthalten, welche für das externe Model-Tool benötigt werden
		(siehe ReadMe.txt im Ordner).

	Der Vorteil dieses OpcUa-Konzepts ist, dass damit benutzerdefinierte Hierarchien im Address-Raum möglich sind,
	die Funktionalität hinter den einzelnen Knoten aber ganz einfach über das bereits bestehende B&R-Modell
	abgebildet werden kann.
	Ebenso können von anderen Institutionen zur Verfügung gestellte Modelle ganz einfach verwendet werden, z.B. das
	Modell einer von der Opc-Foundation erstellten Companion Specification. Solche CS werden von der Opc-Foundation
	in Zusammenarbeit mit Industrie-Verbänden und Dach-Institutionen erstellt und haben das Ziel, die Schnittstelle
	bestimmter Maschinen international zu standardisieren.
	Es sind mittlerweile sehr viele solcher Companion Specifications und deren Modelle erhältlich. Z.B. gibt es für
	Injektions-Maschinen die Companion Specification 'EuroMap' sowie die zugehörigen Modelle.
```

### ReadMe.txt
```
In diesem Ordner sind die Dateien enthalten, welche für das externe Model-Tool 'UaModeler' benötigt werden:

	OpcUa_MyMachine.pdf								Exemplarische Anleitung zum Erzeugen eines eigenen Daten-Modells (Entwurf)
																		unter AS4.6.

	aircondmodel.tt2pro								Projekt-Datei für das Modeler-Tool 'UaModeler'.

	aircondmodel.xml									Vom Modeler exportierte Datei, welche das neue Modell enthält.
																			Sie wurde in die Configuration View	unter "Connectivity/OpcUa" kopiert und
																			in "*.uanodeset" umbenannt.
																			Damit wurde das neue Modell ins AS importiert.

	aircondmodel.ua										Vom Modeler erzeugte Datei, die intern benötigt wird.
	aircondmodel.bsd									Vom Modeler exportierte Datei, welche das Binär-Schema enthält.
	aircondmodel.xsd									Vom Modeler exportierte Datei, welche das XML-Schema enthält.
```

- aircondmodel.tt2pro (not shown)

- aircondmodel.ua (binary file, 41684 bytes)
- aircondmodel.bsd (not shown)

- aircondmodel.xsd (not shown)

### G_AirCond.typ - Package data types
```iecst
TYPE
	AirCond_TYP : 	STRUCT  (*Daten einer Klima-Anlage*)
		sName : STRING[32]; (*Name der Instanz*)
		Act : AirCondAct_TYP; (*Ist-Werte*)
		Set : AirCondSet_TYP; (*Soll-Werte*)
	END_STRUCT;
	AirCondAct_TYP : 	STRUCT  (*Ist-Werte*)
		eOperationMode : AirCondOperationMode_ENUM; (*Betriebs-Modus*)
		rTemperature : REAL; (*Temperatur in [°C]*)
		nFanLevel : USINT; (*Lüfter-Stufe 0-5; 0=Off*)
	END_STRUCT;
	AirCondOperationMode_ENUM :
		( (*Betriebs-Modus*)
		eAC_OPERATIONMODE_OFF, (*Aus*)
		eAC_OPERATIONMODE_MANUAL, (*Manuell*)
		eAC_OPERATIONMODE_AUTO (*Automatik*)
		);
	AirCondSet_TYP : 	STRUCT  (*Sollwerte*)
		rTemperature : REAL; (*Temperatur in [°C] für Automatik*)
		nFanLevel : USINT; (*Lüfter-Stufe 0-5 für Manuell*)
	END_STRUCT;
	AirCondIntern_TYP : 	STRUCT  (*Interne Daten für Klima-Anlage*)
		rDiff : REAL; (*Differenz zwischen Soll- und Ist-Temperatur in [°C]*)
		rDiffPercent : REAL; (*Differenz zwischen Soll- und Ist-Temperatur in %*)
		rCoolStepTemp : REAL; (*Simulations-Dekrement zur Kühlung in [°C]*)
		MethSetOperationMode : AirCondIntMethSetOpMode_TYP; (*Daten für SetOperationMode*)
		EvntOperationModeChanged : AirCondIntEvntOpModeChanged_TYP;
	END_STRUCT;
	AirCondIntMethSetOpMode_TYP : 	STRUCT  (*Daten für SetOperationMode*)
		nStep : UINT; (*Schritt für die Schrittkette*)
		fbUaSrv_MethodOperate : UaSrv_MethodOperate; (*Funktionsblock zum Behandeln der Methode*)
		ArgsIn : AirCondIntMethSetOpModeIn_TYP; (*Eingangs-Argumente*)
		ArgsOut : AirCondIntMethSetOpModeOut_TYP; (*Ausgangs-Argumente*)
	END_STRUCT;
	AirCondIntMethSetOpModeIn_TYP : 	STRUCT  (*Eingangs-Argumente für SetOperationMode*)
		eOperationMode : AirCondOperationMode_ENUM; (*Betriebs-Modus*)
	END_STRUCT;
	AirCondMethodStatus_ENUM :
		( (*Applikations-Status für SetOperationMode*)
		eAC_METH_STATUS_OK, (*Ok*)
		eAC_METH_STATUS_INVALID_OPMODE (*Betriebs-Modus ist nicht gültig*)
		);
	AirCondIntMethSetOpModeOut_TYP : 	STRUCT  (*Ausgangs-Argumente für SetOperationMode*)
		eStatus : AirCondMethodStatus_ENUM; (*Status*)
	END_STRUCT;
	AirCondIntEvntOpModeChanged_TYP : 	STRUCT
		nStep : UINT; (*Schritt für die Schrittkette*)
		eOldOperationMode : AirCondOperationMode_ENUM; (*Betriebs-Modus*)
		bFire : BOOL; (*Kommando zum Feuern des Events*)
		fbUaSrv_GetNamespaceIndex : UaSrv_GetNamespaceIndex; (*Funktionsblock zum Ermitteln eines NamespaceIndex*)
		nNamespaceIndexAirCond : UINT; (*NamespaceIndex  des eigenen Modells*)
		sNamespaceIndexAirCond : STRING[3]; (*NamespaceIndex  des eigenen Modells*)
		sEventFieldsBaseVarName : STRING[128]; (*Beginn des Variablennamens zu den Feld-Werten*)
		sEventFieldSourceNode : STRING[64]; (*Numerische NodeId des Hauptknotens*)
		fbUaSrv_FireEvent : UaSrv_FireEvent; (*Funktionsblock zum Feuern des Events*)
		Fields : AirCondIntEvntOmcFields_TYP; (*Felder des Events*)
	END_STRUCT;
	AirCondIntEvntOmcFields_TYP : 	STRUCT  (*Felder des Events*)
		SourceNode : UANodeID;
		Message : UALocalizedText; (*Wert des Felds 'Message'*)
		OldOperationMode : AirCondOperationMode_ENUM; (*Wert des Felds 'OldOperationMode'*)
		NewOperationMode : AirCondOperationMode_ENUM; (*Wert des Felds 'NewOperationMode'*)
		FieldCfg : ARRAY[0..nAIR_COND_EVENT_FIELD_INDEX_MAX]OF UaSrv_FireEventFieldType; (*Konfiguration der Felder*)
	END_STRUCT;
END_TYPE
```

### G_AirCond.var - Package variables
```iecst
VAR CONSTANT
	rAIR_COND_TEMP_MIN : REAL := 15.0;
	rAIR_COND_TEMP_OUTSIDE : REAL := 26.0;
	nAIR_COND_EVENT_FIELD_INDEX_MAX : UINT := 3;
END_VAR
```

### Program Logical/Tasks/AirCond/AirCondC/AirCondC (ANSIC) - Klima-Anlagen: Eigenes Daten-Modell

#### AirCondC.c - Implementation code
```c
#include <bur/plctypes.h>

#ifdef _DEFAULT_INCLUDES
	#include <AsDefault.h>
#endif

// NOLINTBEGIN(readability-*, bugprone-easily-swappable-parameters, bugprone-branch-clone, clang-diagnostic-invalid-utf8, clang-diagnostic-invalid-source-encoding, clang-diagnostic-pointer-arith, clang-diagnostic-strict-prototypes, clang-diagnostic-shadow, clang-diagnostic-bad-function-cast, clang-analyzer-security.insecureAPI.*, hicpp-uppercase-literal-suffix, hicpp-function-size, cppcoreguidelines-*, performance-*)

// Prototypen
void InitAirCond(AirCond_TYP* pInstance, AirCondIntern_TYP* pIntern, STRING* pInstanceName, STRING* pMethodName, STRING* pEventFieldsBaseVarName, STRING* pEventFieldSourceNode);
void OperateAirCond(AirCond_TYP* pInstance, AirCondIntern_TYP* pIntern);
void SimulateAirCond(AirCond_TYP* pInstance, AirCondIntern_TYP* pIntern);
void GetOperationModeText(AirCondOperationMode_ENUM eOperationMode, STRING* pText);

void _INIT Init(void)
{
	// Initialisierung der einzelnen Instanzen
	InitAirCond(&AirCond_BedRoom, &AirCondIntern_BedRoom, "Bed room", "BedRoomSetOperationMode", "AirCondC:AirCondIntern_BedRoom.EvntOperationModeChanged.Fields", "5013");
	InitAirCond(&AirCond_Corridor, &AirCondIntern_Corridor, "Corridor", "CorridorSetOperationMode", "AirCondC:AirCondIntern_Corridor.EvntOperationModeChanged.Fields", "5017");
	InitAirCond(&AirCond_LivingRoom, &AirCondIntern_LivingRoom, "Living room", "LivingRoomSetOperationMode", "AirCondC:AirCondIntern_LivingRoom.EvntOperationModeChanged.Fields", "5020");

}

void _CYCLIC Cyclic(void)
{
	// Steuerung und Simulation der einzelnen Instanzen
	OperateAirCond(&AirCond_BedRoom, &AirCondIntern_BedRoom);
	OperateAirCond(&AirCond_Corridor, &AirCondIntern_Corridor);
	OperateAirCond(&AirCond_LivingRoom, &AirCondIntern_LivingRoom);
}

void _EXIT Exit(void)
{
}

// Initialisierung einer Instanz
void InitAirCond(AirCond_TYP* pInstance, AirCondIntern_TYP* pIntern, STRING* pInstanceName, STRING* pMethodName, STRING* pEventFieldsBaseVarName, STRING* pEventFieldSourceNode)
{
	// Logik
	pInstance->Act.eOperationMode = eAC_OPERATIONMODE_OFF;
	pInstance->Act.rTemperature = rAIR_COND_TEMP_OUTSIDE;
	pInstance->Act.nFanLevel = 0;
	pInstance->Set.rTemperature = 20.0f;
	pInstance->Set.nFanLevel = 0;

	// Name der Instanz
	brsstrcpy((UDINT)&pInstance->sName, (UDINT)pInstanceName);

	// Methode 'SetOperationMode'
	brsstrcpy((UDINT)&pIntern->MethSetOperationMode.fbUaSrv_MethodOperate.MethodName, (UDINT)pMethodName);

	// Event 'AirConditionOperationModeChanged'
	brsstrcpy((UDINT)&pIntern->EvntOperationModeChanged.sEventFieldsBaseVarName, (UDINT)pEventFieldsBaseVarName);
	brsstrcpy((UDINT)&pIntern->EvntOperationModeChanged.sEventFieldSourceNode, (UDINT)pEventFieldSourceNode);

}

// Steuerung einer Instanz
void OperateAirCond(AirCond_TYP* pInstance, AirCondIntern_TYP* pIntern)
{
	// Methode 'SetOperationMode'
	switch(pIntern->MethSetOperationMode.nStep)
	{
		case 0:
			// Prüfen, ob Methode von einem Client aufgerufen wurde
			pIntern->MethSetOperationMode.fbUaSrv_MethodOperate.Execute = 1;
			pIntern->MethSetOperationMode.fbUaSrv_MethodOperate.Action = UaMoa_CheckIsCalled;
			if(pIntern->MethSetOperationMode.fbUaSrv_MethodOperate.Done == 1)
			{
				pIntern->MethSetOperationMode.fbUaSrv_MethodOperate.Execute = 0;
				if(pIntern->MethSetOperationMode.fbUaSrv_MethodOperate.IsCalled == 1)
				{
					// Variablen der Eingans-Argumente sind besetzt -> Methode ausführen
					pIntern->MethSetOperationMode.nStep = 1;
				}
			}
			else if(pIntern->MethSetOperationMode.fbUaSrv_MethodOperate.Error == 1)
			{
				// Fehler, aber trotzdem weiter machen
				pIntern->MethSetOperationMode.fbUaSrv_MethodOperate.Execute = 0;
			}
			break;

		case 1:
			// Ausführen der Methode
			if(pIntern->MethSetOperationMode.ArgsIn.eOperationMode >= eAC_OPERATIONMODE_OFF && pIntern->MethSetOperationMode.ArgsIn.eOperationMode <= eAC_OPERATIONMODE_AUTO)
			{
				pInstance->Act.eOperationMode = pIntern->MethSetOperationMode.ArgsIn.eOperationMode;
				pIntern->MethSetOperationMode.ArgsOut.eStatus = eAC_METH_STATUS_OK;
			}
			else
			{
				pIntern->MethSetOperationMode.ArgsOut.eStatus = eAC_METH_STATUS_INVALID_OPMODE;
			}
			pIntern->MethSetOperationMode.nStep = 2;
			break;

		case 2:
			// Rückmelden, dass Methode ausgeführt wurde. Zu diesem Zeitpunkt müssen die Ausgangs-Argumente besetzt sein und dürfen nicht mehr geändert werden
			pIntern->MethSetOperationMode.fbUaSrv_MethodOperate.Execute = 1;
			pIntern->MethSetOperationMode.fbUaSrv_MethodOperate.Action = UaMoa_Finished;
			if(pIntern->MethSetOperationMode.fbUaSrv_MethodOperate.Done == 1)
			{
				pIntern->MethSetOperationMode.fbUaSrv_MethodOperate.Execute = 0;
				pIntern->MethSetOperationMode.nStep = 0;
			}
			else if(pIntern->MethSetOperationMode.fbUaSrv_MethodOperate.Error == 1)
			{
				// Fehler, aber trotzdem weiter machen
				pIntern->MethSetOperationMode.fbUaSrv_MethodOperate.Execute = 0;
				pIntern->MethSetOperationMode.nStep = 0;
			}
			break;

	}
	UaSrv_MethodOperate(&pIntern->MethSetOperationMode.fbUaSrv_MethodOperate);

	// Begrenzung der SetTemp
	if(pInstance->Set.rTemperature < rAIR_COND_TEMP_MIN)
	{
		pInstance->Set.rTemperature = rAIR_COND_TEMP_MIN;
	}
	else if(pInstance->Set.rTemperature > rAIR_COND_TEMP_OUTSIDE)
	{
		pInstance->Set.rTemperature = rAIR_COND_TEMP_OUTSIDE;
	}
	// Berechnung der internen Werte (Abweichung in Prozent)
	pIntern->rDiff = pInstance->Act.rTemperature - pInstance->Set.rTemperature;
	pIntern->rDiffPercent = pIntern->rDiff / pInstance->Act.rTemperature * 100.0f;
	// Steuern des Lüfters
	if(pInstance->Act.eOperationMode == eAC_OPERATIONMODE_OFF)
	{
		// Lüfter ausschalten
		pInstance->Act.nFanLevel = 0;
	}
	else if(pInstance->Act.eOperationMode == eAC_OPERATIONMODE_MANUAL)
	{
		// Lüfter-Stufe aus manueller Vorgabe übernehmen
		if(pInstance->Set.nFanLevel > 5)
		{
			pInstance->Act.nFanLevel = 5;
		}
		else
		{
			pInstance->Act.nFanLevel = pInstance->Set.nFanLevel;
		}
	}
	else if(pInstance->Act.eOperationMode == eAC_OPERATIONMODE_AUTO)
	{
		// Lüfter-Stufe je nach Temperatur-Differenz setzen
		if(pIntern->rDiffPercent <= 0.0f)
		{
			pInstance->Act.nFanLevel = 0;
		}
		else if(pIntern->rDiffPercent <= 10.0f)
		{
			pInstance->Act.nFanLevel = 1;
		}
		else if(pIntern->rDiffPercent <= 15.0f)
		{
			pInstance->Act.nFanLevel = 2;
		}
		else if(pIntern->rDiffPercent <= 20.0f)
		{
			pInstance->Act.nFanLevel = 3;
		}
		else if(pIntern->rDiffPercent <= 25.0f)
		{
			pInstance->Act.nFanLevel = 4;
		}
		else
		{
			pInstance->Act.nFanLevel = 5;
		}
	}
	SimulateAirCond(pInstance, pIntern);

	// Event 'AirConditionOperationModeChanged'
	if(pInstance->Act.eOperationMode != pIntern->EvntOperationModeChanged.eOldOperationMode)
	{
		// Besetzen der Felder mit aktuellen Werten
		pIntern->EvntOperationModeChanged.Fields.OldOperationMode = pIntern->EvntOperationModeChanged.eOldOperationMode;
		pIntern->EvntOperationModeChanged.Fields.NewOperationMode = pInstance->Act.eOperationMode;
		STRING sMessageText[512];
		brsmemset((UDINT)&sMessageText, 0, sizeof(sMessageText));
		brsstrcpy((UDINT)&sMessageText, (UDINT)&"Operation mode of air condition '");
		brsstrcat((UDINT)&sMessageText, (UDINT)&pInstance->sName);
		brsstrcat((UDINT)&sMessageText, (UDINT)&"' has changed from '");
		GetOperationModeText(pIntern->EvntOperationModeChanged.Fields.OldOperationMode, sMessageText);
		brsstrcat((UDINT)&sMessageText, (UDINT)&"' to '");
		GetOperationModeText(pIntern->EvntOperationModeChanged.Fields.NewOperationMode, sMessageText);
		brsstrcat((UDINT)&sMessageText, (UDINT)&"' (C).");
		brsstrcpy((UDINT)&pIntern->EvntOperationModeChanged.Fields.Message.Text, (UDINT)&sMessageText);
		// Event feuern
		pIntern->EvntOperationModeChanged.bFire = 1;
	}
	pIntern->EvntOperationModeChanged.eOldOperationMode = pInstance->Act.eOperationMode;
	switch(pIntern->EvntOperationModeChanged.nStep)
	{
		case 0:
			// Ermitteln des Namespace-Index für Fremdmodell-Adressbereich am am B&R-Server
			pIntern->EvntOperationModeChanged.fbUaSrv_GetNamespaceIndex.Execute = 1;
			brsstrcpy((UDINT)&pIntern->EvntOperationModeChanged.fbUaSrv_GetNamespaceIndex.NamespaceUri, (UDINT)&"http://br-automation.com/AirCondModel/");
			if(pIntern->EvntOperationModeChanged.fbUaSrv_GetNamespaceIndex.Done == 1)
			{
				pIntern->EvntOperationModeChanged.fbUaSrv_GetNamespaceIndex.Execute = 0;
				pIntern->EvntOperationModeChanged.nNamespaceIndexAirCond = pIntern->EvntOperationModeChanged.fbUaSrv_GetNamespaceIndex.NamespaceIndex;
				brsitoa((DINT)pIntern->EvntOperationModeChanged.nNamespaceIndexAirCond, (UDINT)&pIntern->EvntOperationModeChanged.sNamespaceIndexAirCond);
				pIntern->EvntOperationModeChanged.nStep += 1;
			}
			else if(pIntern->EvntOperationModeChanged.fbUaSrv_GetNamespaceIndex.Error == 1)
			{
				// Fehler
				pIntern->EvntOperationModeChanged.fbUaSrv_GetNamespaceIndex.Execute = 0;
			}
			break;

		case 1:
			// Initialisierung zum Feuern des Events
			// Event-Typ
			pIntern->EvntOperationModeChanged.fbUaSrv_FireEvent.EventType.NamespaceIndex = pIntern->EvntOperationModeChanged.nNamespaceIndexAirCond;
			pIntern->EvntOperationModeChanged.fbUaSrv_FireEvent.EventType.IdentifierType = UAIdentifierType_Numeric;
			brsstrcpy((UDINT)&pIntern->EvntOperationModeChanged.fbUaSrv_FireEvent.EventType.Identifier, (UDINT)&"1002"); // = AirConditionOperationModeChanged
			// Event-Felder
			UINT nFieldIndex = 0;
			STRING sFieldNameTotal[128];
			brsmemset((UDINT)&sFieldNameTotal, 0, sizeof(sFieldNameTotal));
			STRING sVarNameTotal[255];
			brsmemset((UDINT)&sVarNameTotal, 0, sizeof(sVarNameTotal));
			// SourceNode
			brsstrcpy((UDINT)&pIntern->EvntOperationModeChanged.Fields.FieldCfg[nFieldIndex].BrowsePath, (UDINT)&"/SourceNode");
			brsstrcpy((UDINT)&sVarNameTotal, (UDINT)pIntern->EvntOperationModeChanged.sEventFieldsBaseVarName);
			brsstrcat((UDINT)&sVarNameTotal, (UDINT)&".SourceNode");
			brsstrcpy((UDINT)&pIntern->EvntOperationModeChanged.Fields.FieldCfg[nFieldIndex].Variable, (UDINT)&sVarNameTotal);
			pIntern->EvntOperationModeChanged.Fields.SourceNode.NamespaceIndex = pIntern->EvntOperationModeChanged.nNamespaceIndexAirCond;
			pIntern->EvntOperationModeChanged.Fields.SourceNode.IdentifierType = UAIdentifierType_Numeric;
			brsstrcpy((UDINT)&pIntern->EvntOperationModeChanged.Fields.SourceNode.Identifier, (UDINT)&pIntern->EvntOperationModeChanged.sEventFieldSourceNode);
			// Message
			nFieldIndex += 1;
			brsstrcpy((UDINT)&pIntern->EvntOperationModeChanged.Fields.FieldCfg[nFieldIndex].BrowsePath, (UDINT)&"/Message");
			brsstrcpy((UDINT)&sVarNameTotal, (UDINT)pIntern->EvntOperationModeChanged.sEventFieldsBaseVarName);
			brsstrcat((UDINT)&sVarNameTotal, (UDINT)&".Message");
			brsstrcpy((UDINT)&pIntern->EvntOperationModeChanged.Fields.FieldCfg[nFieldIndex].Variable, (UDINT)&sVarNameTotal);
			brsstrcpy((UDINT)&pIntern->EvntOperationModeChanged.Fields.Message.Text, (UDINT)&"Operation mode has changed.");
			// OldOperationMode
			nFieldIndex += 1;
			brsstrcpy((UDINT)&sFieldNameTotal, (UDINT)&"/");
			brsstrcat((UDINT)&sFieldNameTotal, (UDINT)pIntern->EvntOperationModeChanged.sNamespaceIndexAirCond);
			brsstrcat((UDINT)&sFieldNameTotal, (UDINT)&":OldOperationMode");
			brsstrcpy((UDINT)&pIntern->EvntOperationModeChanged.Fields.FieldCfg[nFieldIndex].BrowsePath, (UDINT)&sFieldNameTotal);
			brsstrcpy((UDINT)&sVarNameTotal, (UDINT)pIntern->EvntOperationModeChanged.sEventFieldsBaseVarName);
			brsstrcat((UDINT)&sVarNameTotal, (UDINT)&".OldOperationMode");
			brsstrcpy((UDINT)&pIntern->EvntOperationModeChanged.Fields.FieldCfg[nFieldIndex].Variable, (UDINT)&sVarNameTotal);
			// NewOperationMode
			nFieldIndex += 1;
			brsstrcpy((UDINT)&sFieldNameTotal, (UDINT)&"/");
			brsstrcat((UDINT)&sFieldNameTotal, (UDINT)pIntern->EvntOperationModeChanged.sNamespaceIndexAirCond);
			brsstrcat((UDINT)&sFieldNameTotal, (UDINT)&":NewOperationMode");
			brsstrcpy((UDINT)&pIntern->EvntOperationModeChanged.Fields.FieldCfg[nFieldIndex].BrowsePath, (UDINT)&sFieldNameTotal);
			brsstrcpy((UDINT)&sVarNameTotal, (UDINT)pIntern->EvntOperationModeChanged.sEventFieldsBaseVarName);
			brsstrcat((UDINT)&sVarNameTotal, (UDINT)&".NewOperationMode");
			brsstrcpy((UDINT)&pIntern->EvntOperationModeChanged.Fields.FieldCfg[nFieldIndex].Variable, (UDINT)&sVarNameTotal);
			// Statische Funktionsblock-Eingänge
			pIntern->EvntOperationModeChanged.fbUaSrv_FireEvent.EventFieldCount = nFieldIndex+1;
			pIntern->EvntOperationModeChanged.fbUaSrv_FireEvent.EventFields = (UaSrv_FireEventFieldType*)&pIntern->EvntOperationModeChanged.Fields.FieldCfg;
			pIntern->EvntOperationModeChanged.nStep += 1;
			break;

		case 2:
			// Prüfen, ob Event gefeuert werden muss
			if(pIntern->EvntOperationModeChanged.bFire == 1)
			{
				pIntern->EvntOperationModeChanged.bFire = 0;
				pIntern->EvntOperationModeChanged.nStep += 1;
			}
			break;

		case 3:
			// Event feuern
			pIntern->EvntOperationModeChanged.fbUaSrv_FireEvent.Execute = 1;
			if(pIntern->EvntOperationModeChanged.fbUaSrv_FireEvent.Done == 1)
			{
				pIntern->EvntOperationModeChanged.fbUaSrv_FireEvent.Execute = 0;
				pIntern->EvntOperationModeChanged.nStep -= 1;
			}
			else if(pIntern->EvntOperationModeChanged.fbUaSrv_FireEvent.Error == 1)
			{
				// Fehler
			}
			break;

	}
	UaSrv_GetNamespaceIndex(&pIntern->EvntOperationModeChanged.fbUaSrv_GetNamespaceIndex);
	UaSrv_FireEvent(&pIntern->EvntOperationModeChanged.fbUaSrv_FireEvent);
}

// Simulation einer Instanz (Verändern der ActTemp)
void SimulateAirCond(AirCond_TYP* pInstance, AirCondIntern_TYP* pIntern)
{
	// Stetiges Angleichen an die Aussentemperatur
	pInstance->Act.rTemperature = pInstance->Act.rTemperature + 0.0005f;
	if(pInstance->Act.rTemperature > rAIR_COND_TEMP_OUTSIDE)
	{
		pInstance->Act.rTemperature = rAIR_COND_TEMP_OUTSIDE;
	}
	// Kühlen
	if(pInstance->Act.eOperationMode != eAC_OPERATIONMODE_OFF)
	{
		// Je nach Lüfter-Stufe kühlt die ActTemp runter
		pIntern->rCoolStepTemp = (REAL)pInstance->Act.nFanLevel * 0.005f;
		pInstance->Act.rTemperature = pInstance->Act.rTemperature - pIntern->rCoolStepTemp;
	}
	// Physikalische Begrenzung der ActTemp
	if(pInstance->Act.rTemperature < rAIR_COND_TEMP_MIN)
	{
		pInstance->Act.rTemperature = rAIR_COND_TEMP_MIN;
	}
}

// Wandeln des Betriebsmodus in Text
void GetOperationModeText(AirCondOperationMode_ENUM eOperationMode, STRING* pText)
{
	if(eOperationMode == eAC_OPERATIONMODE_OFF)
	{
		brsstrcat((UDINT)pText, (UDINT)&"Off");
	}
	else if(eOperationMode == eAC_OPERATIONMODE_MANUAL)
	{
		brsstrcat((UDINT)pText, (UDINT)&"Manual");
	}
	else if(eOperationMode == eAC_OPERATIONMODE_AUTO)
	{
		brsstrcat((UDINT)pText, (UDINT)&"Automatic");
	}
	else
	{
		brsstrcat((UDINT)pText, (UDINT)&"Unknown");
	}
}

// NOLINTEND(readability-*, bugprone-easily-swappable-parameters, bugprone-branch-clone, clang-diagnostic-invalid-utf8, clang-diagnostic-invalid-source-encoding, clang-diagnostic-pointer-arith, clang-diagnostic-strict-prototypes, clang-diagnostic-shadow, clang-diagnostic-bad-function-cast, clang-analyzer-security.insecureAPI.*, hicpp-uppercase-literal-suffix, hicpp-function-size, cppcoreguidelines-*, performance-*)
```

#### AirCondC.var - Local variables
```iecst
VAR
	AirCond_BedRoom : AirCond_TYP;
	AirCondIntern_BedRoom : AirCondIntern_TYP;
	AirCond_Corridor : AirCond_TYP;
	AirCondIntern_Corridor : AirCondIntern_TYP;
	AirCond_LivingRoom : AirCond_TYP;
	AirCondIntern_LivingRoom : AirCondIntern_TYP;
END_VAR
```

- Methods.uam (not shown)

### Program Logical/Tasks/AirCond/AirCondST/AirCondST (IEC) - Klima-Anlagen: Eigenes Daten-Modell

#### AirCondST.st - Init, cyclic, exit code
```iecst
PROGRAM _INIT
	// Initialisierung der einzelnen Instanzen
	pInstance ACCESS ADR(AirCond_BedRoom);
	pIntern ACCESS ADR(AirCondIntern_BedRoom);
	InitAirCond;
	pInstance.sName := 'Bed room';
	pIntern.MethSetOperationMode.fbUaSrv_MethodOperate.MethodName := 'BedRoomSetOperationMode';
	pIntern.EvntOperationModeChanged.sEventFieldsBaseVarName := 'AirCondST:AirCondIntern_BedRoom.EvntOperationModeChanged.Fields';
	pIntern.EvntOperationModeChanged.sEventFieldSourceNode := '5023';

	pInstance ACCESS ADR(AirCond_Corridor);
	pIntern ACCESS ADR(AirCondIntern_Corridor);
	InitAirCond;
	pInstance.sName := 'Corridor';
	pIntern.MethSetOperationMode.fbUaSrv_MethodOperate.MethodName := 'CorridorSetOperationMode';
	pIntern.EvntOperationModeChanged.sEventFieldsBaseVarName := 'AirCondST:AirCondIntern_Corridor.EvntOperationModeChanged.Fields';
	pIntern.EvntOperationModeChanged.sEventFieldSourceNode := '5027';

	pInstance ACCESS ADR(AirCond_LivingRoom);
	pIntern ACCESS ADR(AirCondIntern_LivingRoom);
	InitAirCond;
	pInstance.sName := 'Living room';
	pIntern.MethSetOperationMode.fbUaSrv_MethodOperate.MethodName := 'LivingRoomSetOperationMode';
	pIntern.EvntOperationModeChanged.sEventFieldsBaseVarName := 'AirCondST:AirCondIntern_LivingRoom.EvntOperationModeChanged.Fields';
	pIntern.EvntOperationModeChanged.sEventFieldSourceNode := '5030';
END_PROGRAM

PROGRAM _CYCLIC
	// Steuerung und Simulation der einzelnen Instanzen
	pInstance ACCESS ADR(AirCond_BedRoom);
	pIntern ACCESS ADR(AirCondIntern_BedRoom);
	OperateAirCond;
	pInstance ACCESS ADR(AirCond_Corridor);
	pIntern ACCESS ADR(AirCondIntern_Corridor);
	OperateAirCond;
	pInstance ACCESS ADR(AirCond_LivingRoom);
	pIntern ACCESS ADR(AirCondIntern_LivingRoom);
	OperateAirCond;
END_PROGRAM

PROGRAM _EXIT
END_PROGRAM
```

#### AirCondST.var - Local variables
```iecst
VAR
	AirCond_BedRoom : AirCond_TYP;
	AirCondIntern_BedRoom : AirCondIntern_TYP;
	AirCond_Corridor : AirCond_TYP;
	AirCondIntern_Corridor : AirCondIntern_TYP;
	AirCond_LivingRoom : AirCond_TYP;
	AirCondIntern_LivingRoom : AirCondIntern_TYP;
	pInstance : REFERENCE TO AirCond_TYP;
	pIntern : REFERENCE TO AirCondIntern_TYP;
	sMessageText : STRING[512];
	eOperationMode : AirCondOperationMode_ENUM;
	sOperationModeText : STRING[512];
	nFieldIndex : UINT;
	sFieldNameTotal : STRING[128];
	sVarNameTotal : STRING[256];
END_VAR
```
